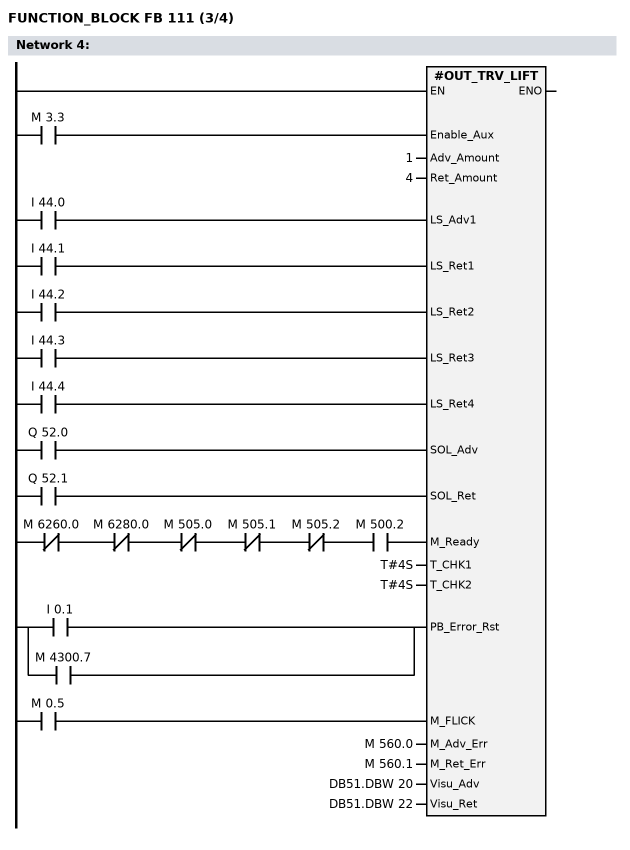

      A     M      3.3;
      =     L      0.0;
      BLD   103;
      A     I     44.0;
      =     L      0.1;
      BLD   103;
      A     I     44.1;
      =     L      0.2;
      BLD   103;
      A     I     44.2;
      =     L      0.4;
      BLD   103;
      A     I     44.3;
      =     L      0.6;
      BLD   103;
      A     I     44.4;
      =     L      1.0;
      BLD   103;
      A     Q     52.0;
      =     L      1.1;
      BLD   103;
      A     Q     52.1;
      =     L      1.2;
      BLD   103;
      AN    M   6260.0;
      AN    M   6280.0;
      AN    M    505.0;
      AN    M    505.1;
      AN    M    505.2;
      A     M    500.2;
      =     L      1.3;
      BLD   103;
      A(    ;
      O     I      0.1;
      O     M   4300.7;
      )     ;
      =     L      1.5;
      BLD   103;
      A     M      0.5;
      =     L      1.6;
      BLD   103;
      CALL #OUT_TRV_LIFT (
           Enable_Aux               := L      0.0,
           Adv_Amount               := 1,
           Ret_Amount               := 4,
           LS_Adv1                  := L      0.1,
           LS_Ret1                  := L      0.2,
           LS_Ret2                  := L      0.4,
           LS_Ret3                  := L      0.6,
           LS_Ret4                  := L      1.0,
           SOL_Adv                  := L      1.1,
           SOL_Ret                  := L      1.2,
           M_Ready                  := L      1.3,
           T_CHK1                   := T#4S,
           T_CHK2                   := T#4S,
           PB_Error_Rst             := L      1.5,
           M_FLICK                  := L      1.6,
           M_Adv_Err                := M    560.0,
           M_Ret_Err                := M    560.1,
           Visu_Adv                 := DB51.DBW   20,
           Visu_Ret                 := DB51.DBW   22);
      NOP   0;
NETWORK
TITLE =OUT TRV 급전이상 항시OFF
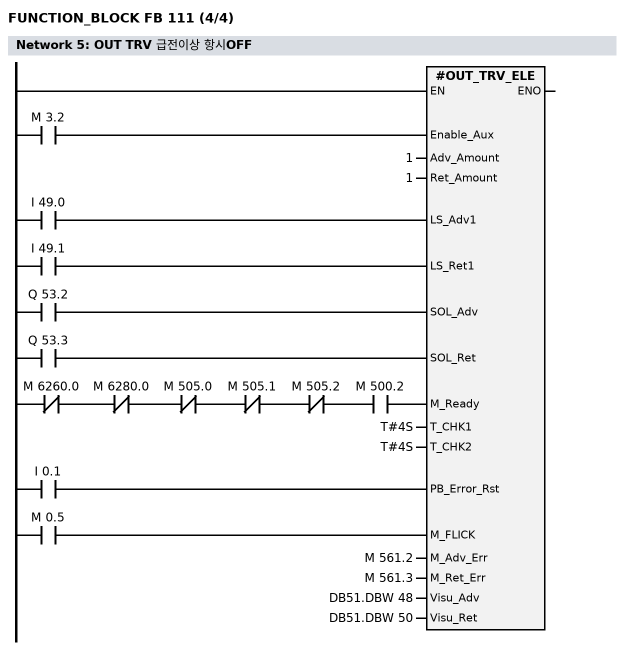

      A     M      3.2;
      =     L      0.0;
      BLD   103;
      A     I     49.0;
      =     L      0.1;
      BLD   103;
      A     I     49.1;
      =     L      0.2;
      BLD   103;
      A     Q     53.2;
      =     L      1.1;
      BLD   103;
      A     Q     53.3;
      =     L      1.2;
      BLD   103;
      AN    M   6260.0;
      AN    M   6280.0;
      AN    M    505.0;
      AN    M    505.1;
      AN    M    505.2;
      A     M    500.2;
      =     L      1.3;
      BLD   103;
      A     I      0.1;
      =     L      1.5;
      BLD   103;
      A     M      0.5;
      =     L      1.6;
      BLD   103;
      CALL #OUT_TRV_ELE (
           Enable_Aux               := L      0.0,
           Adv_Amount               := 1,
           Ret_Amount               := 1,
           LS_Adv1                  := L      0.1,
           LS_Ret1                  := L      0.2,
           SOL_Adv                  := L      1.1,
           SOL_Ret                  := L      1.2,
           M_Ready                  := L      1.3,
           T_CHK1                   := T#4S,
           T_CHK2                   := T#4S,
           PB_Error_Rst             := L      1.5,
           M_FLICK                  := L      1.6,
           M_Adv_Err                := M    561.2,
           M_Ret_Err                := M    561.3,
           Visu_Adv                 := DB51.DBW   48,
           Visu_Ret                 := DB51.DBW   50);
      NOP   0;
END_FUNCTION_BLOCK

DATA_BLOCK DB 111
TITLE =
VERSION : 0.0

 FB 111
BEGIN
   OUT_TRV_CUSHION_B.Enable_Aux := FALSE;
   OUT_TRV_CUSHION_B.Adv_Amount := 0;
   OUT_TRV_CUSHION_B.Ret_Amount := 0;
   OUT_TRV_CUSHION_B.LS_Adv1 := FALSE;
   OUT_TRV_CUSHION_B.LS_Ret1 := FALSE;
   OUT_TRV_CUSHION_B.LS_Adv2 := FALSE;
   OUT_TRV_CUSHION_B.LS_Ret2 := FALSE;
   OUT_TRV_CUSHION_B.LS_Adv3 := FALSE;
   OUT_TRV_CUSHION_B.LS_Ret3 := FALSE;
   OUT_TRV_CUSHION_B.LS_Adv4 := FALSE;
   OUT_TRV_CUSHION_B.LS_Ret4 := FALSE;
   OUT_TRV_CUSHION_B.SOL_Adv := FALSE;
   OUT_TRV_CUSHION_B.SOL_Ret := FALSE;
   OUT_TRV_CUSHION_B.M_Ready := FALSE;
   OUT_TRV_CUSHION_B.T_CHK1 := T#0MS;
   OUT_TRV_CUSHION_B.T_CHK2 := T#0MS;
   OUT_TRV_CUSHION_B.PB_Lamp_CHK := FALSE;
   OUT_TRV_CUSHION_B.PB_Error_Rst := FALSE;
   OUT_TRV_CUSHION_B.M_FLICK := FALSE;
   OUT_TRV_CUSHION_B.M_Adv_Err := FALSE;
   OUT_TRV_CUSHION_B.M_Ret_Err := FALSE;
   OUT_TRV_CUSHION_B.LP_Adv := FALSE;
   OUT_TRV_CUSHION_B.LP_Ret := FALSE;
   OUT_TRV_CUSHION_B.Visu_Adv := W#16#0;
   OUT_TRV_CUSHION_B.Visu_Ret := W#16#0;
   OUT_TRV_CUSHION_B.Error_T1.IN := FALSE;
   OUT_TRV_CUSHION_B.Error_T1.PT := T#0MS;
   OUT_TRV_CUSHION_B.Error_T1.Q := FALSE;
   OUT_TRV_CUSHION_B.Error_T1.ET := T#0MS;
   OUT_TRV_CUSHION_B.Error_T1.STATE := B#16#0;
   OUT_TRV_CUSHION_B.Error_T1.STIME := T#0MS;
   OUT_TRV_CUSHION_B.Error_T1.ATIME := T#0MS;
   OUT_TRV_CUSHION_B.Error_T2.IN := FALSE;
   OUT_TRV_CUSHION_B.Error_T2.PT := T#0MS;
   OUT_TRV_CUSHION_B.Error_T2.Q := FALSE;
   OUT_TRV_CUSHION_B.Error_T2.ET := T#0MS;
   OUT_TRV_CUSHION_B.Error_T2.STATE := B#16#0;
   OUT_TRV_CUSHION_B.Error_T2.STIME := T#0MS;
   OUT_TRV_CUSHION_B.Error_T2.ATIME := T#0MS;
   OUT_TRV_CUSHION_B.CHK_Aux1 := FALSE;
   OUT_TRV_CUSHION_B.CHK_Aux2 := FALSE;
   OUT_TRV_CUSHION_B.Error_T1_DN := FALSE;
   OUT_TRV_CUSHION_B.Error_T2_DN := FALSE;
   OUT_TRV_CUSHION_B.Adv_Memo := FALSE;
   OUT_TRV_CUSHION_B.Visu_Adv_Arr[0] := FALSE;
   OUT_TRV_CUSHION_B.Visu_Adv_Arr[1] := FALSE;
   OUT_TRV_CUSHION_B.Visu_Adv_Arr[2] := FALSE;
   OUT_TRV_CUSHION_B.Visu_Adv_Arr[3] := FALSE;
   OUT_TRV_CUSHION_B.Visu_Adv_Arr[4] := FALSE;
   OUT_TRV_CUSHION_B.Visu_Adv_Arr[5] := FALSE;
   OUT_TRV_CUSHION_B.Visu_Adv_Arr[6] := FALSE;
   OUT_TRV_CUSHION_B.Visu_Adv_Arr[7] := FALSE;
   OUT_TRV_CUSHION_B.Visu_Adv_Arr[8] := FALSE;
   OUT_TRV_CUSHION_B.Visu_Adv_Arr[9] := FALSE;
   OUT_TRV_CUSHION_B.Visu_Adv_Arr[10] := FALSE;
   OUT_TRV_CUSHION_B.Visu_Adv_Arr[11] := FALSE;
   OUT_TRV_CUSHION_B.Visu_Adv_Arr[12] := FALSE;
   OUT_TRV_CUSHION_B.Visu_Adv_Arr[13] := FALSE;
   OUT_TRV_CUSHION_B.Visu_Adv_Arr[14] := FALSE;
   OUT_TRV_CUSHION_B.Visu_Adv_Arr[15] := FALSE;
   OUT_TRV_CUSHION_B.Visu_Ret_Arr[0] := FALSE;
   OUT_TRV_CUSHION_B.Visu_Ret_Arr[1] := FALSE;
   OUT_TRV_CUSHION_B.Visu_Ret_Arr[2] := FALSE;
   OUT_TRV_CUSHION_B.Visu_Ret_Arr[3] := FALSE;
   OUT_TRV_CUSHION_B.Visu_Ret_Arr[4] := FALSE;
   OUT_TRV_CUSHION_B.Visu_Ret_Arr[5] := FALSE;
   OUT_TRV_CUSHION_B.Visu_Ret_Arr[6] := FALSE;
   OUT_TRV_CUSHION_B.Visu_Ret_Arr[7] := FALSE;
   OUT_TRV_CUSHION_B.Visu_Ret_Arr[8] := FALSE;
   OUT_TRV_CUSHION_B.Visu_Ret_Arr[9] := FALSE;
   OUT_TRV_CUSHION_B.Visu_Ret_Arr[10] := FALSE;
   OUT_TRV_CUSHION_B.Visu_Ret_Arr[11] := FALSE;
   OUT_TRV_CUSHION_B.Visu_Ret_Arr[12] := FALSE;
   OUT_TRV_CUSHION_B.Visu_Ret_Arr[13] := FALSE;
   OUT_TRV_CUSHION_B.Visu_Ret_Arr[14] := FALSE;
   OUT_TRV_CUSHION_B.Visu_Ret_Arr[15] := FALSE;
   OUT_TRV_CUSHION_B.BLK_Move_Ret := 0;
   OUT_TRV_CUSHION_B.Enable := FALSE;
   OUT_TRV_CUSHION_B.Adv_End := FALSE;
   OUT_TRV_CUSHION_B.Ret_End := FALSE;
   OUT_TRV_GUIDE.Enable_Aux := FALSE;
   OUT_TRV_GUIDE.Adv_Amount := 0;
   OUT_TRV_GUIDE.Ret_Amount := 0;
   OUT_TRV_GUIDE.LS_Adv1 := FALSE;
   OUT_TRV_GUIDE.LS_Ret1 := FALSE;
   OUT_TRV_GUIDE.LS_Adv2 := FALSE;
   OUT_TRV_GUIDE.LS_Ret2 := FALSE;
   OUT_TRV_GUIDE.LS_Adv3 := FALSE;
   OUT_TRV_GUIDE.LS_Ret3 := FALSE;
   OUT_TRV_GUIDE.LS_Adv4 := FALSE;
   OUT_TRV_GUIDE.LS_Ret4 := FALSE;
   OUT_TRV_GUIDE.SOL_Adv := FALSE;
   OUT_TRV_GUIDE.SOL_Ret := FALSE;
   OUT_TRV_GUIDE.M_Ready := FALSE;
   OUT_TRV_GUIDE.T_CHK1 := T#0MS;
   OUT_TRV_GUIDE.T_CHK2 := T#0MS;
   OUT_TRV_GUIDE.PB_Lamp_CHK := FALSE;
   OUT_TRV_GUIDE.PB_Error_Rst := FALSE;
   OUT_TRV_GUIDE.M_FLICK := FALSE;
   OUT_TRV_GUIDE.M_Adv_Err := FALSE;
   OUT_TRV_GUIDE.M_Ret_Err := FALSE;
   OUT_TRV_GUIDE.LP_Adv := FALSE;
   OUT_TRV_GUIDE.LP_Ret := FALSE;
   OUT_TRV_GUIDE.Visu_Adv := W#16#0;
   OUT_TRV_GUIDE.Visu_Ret := W#16#0;
   OUT_TRV_GUIDE.Error_T1.IN := FALSE;
   OUT_TRV_GUIDE.Error_T1.PT := T#0MS;
   OUT_TRV_GUIDE.Error_T1.Q := FALSE;
   OUT_TRV_GUIDE.Error_T1.ET := T#0MS;
   OUT_TRV_GUIDE.Error_T1.STATE := B#16#0;
   OUT_TRV_GUIDE.Error_T1.STIME := T#0MS;
   OUT_TRV_GUIDE.Error_T1.ATIME := T#0MS;
   OUT_TRV_GUIDE.Error_T2.IN := FALSE;
   OUT_TRV_GUIDE.Error_T2.PT := T#0MS;
   OUT_TRV_GUIDE.Error_T2.Q := FALSE;
   OUT_TRV_GUIDE.Error_T2.ET := T#0MS;
   OUT_TRV_GUIDE.Error_T2.STATE := B#16#0;
   OUT_TRV_GUIDE.Error_T2.STIME := T#0MS;
   OUT_TRV_GUIDE.Error_T2.ATIME := T#0MS;
   OUT_TRV_GUIDE.CHK_Aux1 := FALSE;
   OUT_TRV_GUIDE.CHK_Aux2 := FALSE;
   OUT_TRV_GUIDE.Error_T1_DN := FALSE;
   OUT_TRV_GUIDE.Error_T2_DN := FALSE;
   OUT_TRV_GUIDE.Adv_Memo := FALSE;
   OUT_TRV_GUIDE.Visu_Adv_Arr[0] := FALSE;
   OUT_TRV_GUIDE.Visu_Adv_Arr[1] := FALSE;
   OUT_TRV_GUIDE.Visu_Adv_Arr[2] := FALSE;
   OUT_TRV_GUIDE.Visu_Adv_Arr[3] := FALSE;
   OUT_TRV_GUIDE.Visu_Adv_Arr[4] := FALSE;
   OUT_TRV_GUIDE.Visu_Adv_Arr[5] := FALSE;
   OUT_TRV_GUIDE.Visu_Adv_Arr[6] := FALSE;
   OUT_TRV_GUIDE.Visu_Adv_Arr[7] := FALSE;
   OUT_TRV_GUIDE.Visu_Adv_Arr[8] := FALSE;
   OUT_TRV_GUIDE.Visu_Adv_Arr[9] := FALSE;
   OUT_TRV_GUIDE.Visu_Adv_Arr[10] := FALSE;
   OUT_TRV_GUIDE.Visu_Adv_Arr[11] := FALSE;
   OUT_TRV_GUIDE.Visu_Adv_Arr[12] := FALSE;
   OUT_TRV_GUIDE.Visu_Adv_Arr[13] := FALSE;
   OUT_TRV_GUIDE.Visu_Adv_Arr[14] := FALSE;
   OUT_TRV_GUIDE.Visu_Adv_Arr[15] := FALSE;
   OUT_TRV_GUIDE.Visu_Ret_Arr[0] := FALSE;
   OUT_TRV_GUIDE.Visu_Ret_Arr[1] := FALSE;
   OUT_TRV_GUIDE.Visu_Ret_Arr[2] := FALSE;
   OUT_TRV_GUIDE.Visu_Ret_Arr[3] := FALSE;
   OUT_TRV_GUIDE.Visu_Ret_Arr[4] := FALSE;
   OUT_TRV_GUIDE.Visu_Ret_Arr[5] := FALSE;
   OUT_TRV_GUIDE.Visu_Ret_Arr[6] := FALSE;
   OUT_TRV_GUIDE.Visu_Ret_Arr[7] := FALSE;
   OUT_TRV_GUIDE.Visu_Ret_Arr[8] := FALSE;
   OUT_TRV_GUIDE.Visu_Ret_Arr[9] := FALSE;
   OUT_TRV_GUIDE.Visu_Ret_Arr[10] := FALSE;
   OUT_TRV_GUIDE.Visu_Ret_Arr[11] := FALSE;
   OUT_TRV_GUIDE.Visu_Ret_Arr[12] := FALSE;
   OUT_TRV_GUIDE.Visu_Ret_Arr[13] := FALSE;
   OUT_TRV_GUIDE.Visu_Ret_Arr[14] := FALSE;
   OUT_TRV_GUIDE.Visu_Ret_Arr[15] := FALSE;
   OUT_TRV_GUIDE.BLK_Move_Ret := 0;
   OUT_TRV_GUIDE.Enable := FALSE;
   OUT_TRV_GUIDE.Adv_End := FALSE;
   OUT_TRV_GUIDE.Ret_End := FALSE;
   OUT_TRV_CLAMP.Enable_Aux := FALSE;
   OUT_TRV_CLAMP.Adv_Amount := 0;
   OUT_TRV_CLAMP.Ret_Amount := 0;
   OUT_TRV_CLAMP.LS_Adv1 := FALSE;
   OUT_TRV_CLAMP.LS_Ret1 := FALSE;
   OUT_TRV_CLAMP.LS_Adv2 := FALSE;
   OUT_TRV_CLAMP.LS_Ret2 := FALSE;
   OUT_TRV_CLAMP.LS_Adv3 := FALSE;
   OUT_TRV_CLAMP.LS_Ret3 := FALSE;
   OUT_TRV_CLAMP.LS_Adv4 := FALSE;
   OUT_TRV_CLAMP.LS_Ret4 := FALSE;
   OUT_TRV_CLAMP.SOL_Adv := FALSE;
   OUT_TRV_CLAMP.SOL_Ret := FALSE;
   OUT_TRV_CLAMP.M_Ready := FALSE;
   OUT_TRV_CLAMP.T_CHK1 := T#0MS;
   OUT_TRV_CLAMP.T_CHK2 := T#0MS;
   OUT_TRV_CLAMP.PB_Lamp_CHK := FALSE;
   OUT_TRV_CLAMP.PB_Error_Rst := FALSE;
   OUT_TRV_CLAMP.M_FLICK := FALSE;
   OUT_TRV_CLAMP.M_Adv_Err := FALSE;
   OUT_TRV_CLAMP.M_Ret_Err := FALSE;
   OUT_TRV_CLAMP.LP_Adv := FALSE;
   OUT_TRV_CLAMP.LP_Ret := FALSE;
   OUT_TRV_CLAMP.Visu_Adv := W#16#0;
   OUT_TRV_CLAMP.Visu_Ret := W#16#0;
   OUT_TRV_CLAMP.Error_T1.IN := FALSE;
   OUT_TRV_CLAMP.Error_T1.PT := T#0MS;
   OUT_TRV_CLAMP.Error_T1.Q := FALSE;
   OUT_TRV_CLAMP.Error_T1.ET := T#0MS;
   OUT_TRV_CLAMP.Error_T1.STATE := B#16#0;
   OUT_TRV_CLAMP.Error_T1.STIME := T#0MS;
   OUT_TRV_CLAMP.Error_T1.ATIME := T#0MS;
   OUT_TRV_CLAMP.Error_T2.IN := FALSE;
   OUT_TRV_CLAMP.Error_T2.PT := T#0MS;
   OUT_TRV_CLAMP.Error_T2.Q := FALSE;
   OUT_TRV_CLAMP.Error_T2.ET := T#0MS;
   OUT_TRV_CLAMP.Error_T2.STATE := B#16#0;
   OUT_TRV_CLAMP.Error_T2.STIME := T#0MS;
   OUT_TRV_CLAMP.Error_T2.ATIME := T#0MS;
   OUT_TRV_CLAMP.CHK_Aux1 := FALSE;
   OUT_TRV_CLAMP.CHK_Aux2 := FALSE;
   OUT_TRV_CLAMP.Error_T1_DN := FALSE;
   OUT_TRV_CLAMP.Error_T2_DN := FALSE;
   OUT_TRV_CLAMP.Adv_Memo := FALSE;
   OUT_TRV_CLAMP.Visu_Adv_Arr[0] := FALSE;
   OUT_TRV_CLAMP.Visu_Adv_Arr[1] := FALSE;
   OUT_TRV_CLAMP.Visu_Adv_Arr[2] := FALSE;
   OUT_TRV_CLAMP.Visu_Adv_Arr[3] := FALSE;
   OUT_TRV_CLAMP.Visu_Adv_Arr[4] := FALSE;
   OUT_TRV_CLAMP.Visu_Adv_Arr[5] := FALSE;
   OUT_TRV_CLAMP.Visu_Adv_Arr[6] := FALSE;
   OUT_TRV_CLAMP.Visu_Adv_Arr[7] := FALSE;
   OUT_TRV_CLAMP.Visu_Adv_Arr[8] := FALSE;
   OUT_TRV_CLAMP.Visu_Adv_Arr[9] := FALSE;
   OUT_TRV_CLAMP.Visu_Adv_Arr[10] := FALSE;
   OUT_TRV_CLAMP.Visu_Adv_Arr[11] := FALSE;
   OUT_TRV_CLAMP.Visu_Adv_Arr[12] := FALSE;
   OUT_TRV_CLAMP.Visu_Adv_Arr[13] := FALSE;
   OUT_TRV_CLAMP.Visu_Adv_Arr[14] := FALSE;
   OUT_TRV_CLAMP.Visu_Adv_Arr[15] := FALSE;
   OUT_TRV_CLAMP.Visu_Ret_Arr[0] := FALSE;
   OUT_TRV_CLAMP.Visu_Ret_Arr[1] := FALSE;
   OUT_TRV_CLAMP.Visu_Ret_Arr[2] := FALSE;
   OUT_TRV_CLAMP.Visu_Ret_Arr[3] := FALSE;
   OUT_TRV_CLAMP.Visu_Ret_Arr[4] := FALSE;
   OUT_TRV_CLAMP.Visu_Ret_Arr[5] := FALSE;
   OUT_TRV_CLAMP.Visu_Ret_Arr[6] := FALSE;
   OUT_TRV_CLAMP.Visu_Ret_Arr[7] := FALSE;
   OUT_TRV_CLAMP.Visu_Ret_Arr[8] := FALSE;
   OUT_TRV_CLAMP.Visu_Ret_Arr[9] := FALSE;
   OUT_TRV_CLAMP.Visu_Ret_Arr[10] := FALSE;
   OUT_TRV_CLAMP.Visu_Ret_Arr[11] := FALSE;
   OUT_TRV_CLAMP.Visu_Ret_Arr[12] := FALSE;
   OUT_TRV_CLAMP.Visu_Ret_Arr[13] := FALSE;
   OUT_TRV_CLAMP.Visu_Ret_Arr[14] := FALSE;
   OUT_TRV_CLAMP.Visu_Ret_Arr[15] := FALSE;
   OUT_TRV_CLAMP.BLK_Move_Ret := 0;
   OUT_TRV_CLAMP.Enable := FALSE;
   OUT_TRV_CLAMP.Adv_End := FALSE;
   OUT_TRV_CLAMP.Ret_End := FALSE;
   OUT_TRV_LIFT.Enable_Aux := FALSE;
   OUT_TRV_LIFT.Adv_Amount := 0;
   OUT_TRV_LIFT.Ret_Amount := 0;
   OUT_TRV_LIFT.LS_Adv1 := FALSE;
   OUT_TRV_LIFT.LS_Ret1 := FALSE;
   OUT_TRV_LIFT.LS_Adv2 := FALSE;
   OUT_TRV_LIFT.LS_Ret2 := FALSE;
   OUT_TRV_LIFT.LS_Adv3 := FALSE;
   OUT_TRV_LIFT.LS_Ret3 := FALSE;
   OUT_TRV_LIFT.LS_Adv4 := FALSE;
   OUT_TRV_LIFT.LS_Ret4 := FALSE;
   OUT_TRV_LIFT.SOL_Adv := FALSE;
   OUT_TRV_LIFT.SOL_Ret := FALSE;
   OUT_TRV_LIFT.M_Ready := FALSE;
   OUT_TRV_LIFT.T_CHK1 := T#0MS;
   OUT_TRV_LIFT.T_CHK2 := T#0MS;
   OUT_TRV_LIFT.PB_Lamp_CHK := FALSE;
   OUT_TRV_LIFT.PB_Error_Rst := FALSE;
   OUT_TRV_LIFT.M_FLICK := FALSE;
   OUT_TRV_LIFT.M_Adv_Err := FALSE;
   OUT_TRV_LIFT.M_Ret_Err := FALSE;
   OUT_TRV_LIFT.LP_Adv := FALSE;
   OUT_TRV_LIFT.LP_Ret := FALSE;
   OUT_TRV_LIFT.Visu_Adv := W#16#0;
   OUT_TRV_LIFT.Visu_Ret := W#16#0;
   OUT_TRV_LIFT.Error_T1.IN := FALSE;
   OUT_TRV_LIFT.Error_T1.PT := T#0MS;
   OUT_TRV_LIFT.Error_T1.Q := FALSE;
   OUT_TRV_LIFT.Error_T1.ET := T#0MS;
   OUT_TRV_LIFT.Error_T1.STATE := B#16#0;
   OUT_TRV_LIFT.Error_T1.STIME := T#0MS;
   OUT_TRV_LIFT.Error_T1.ATIME := T#0MS;
   OUT_TRV_LIFT.Error_T2.IN := FALSE;
   OUT_TRV_LIFT.Error_T2.PT := T#0MS;
   OUT_TRV_LIFT.Error_T2.Q := FALSE;
   OUT_TRV_LIFT.Error_T2.ET := T#0MS;
   OUT_TRV_LIFT.Error_T2.STATE := B#16#0;
   OUT_TRV_LIFT.Error_T2.STIME := T#0MS;
   OUT_TRV_LIFT.Error_T2.ATIME := T#0MS;
   OUT_TRV_LIFT.CHK_Aux1 := FALSE;
   OUT_TRV_LIFT.CHK_Aux2 := FALSE;
   OUT_TRV_LIFT.Error_T1_DN := FALSE;
   OUT_TRV_LIFT.Error_T2_DN := FALSE;
   OUT_TRV_LIFT.Adv_Memo := FALSE;
   OUT_TRV_LIFT.Visu_Adv_Arr[0] := FALSE;
   OUT_TRV_LIFT.Visu_Adv_Arr[1] := FALSE;
   OUT_TRV_LIFT.Visu_Adv_Arr[2] := FALSE;
   OUT_TRV_LIFT.Visu_Adv_Arr[3] := FALSE;
   OUT_TRV_LIFT.Visu_Adv_Arr[4] := FALSE;
   OUT_TRV_LIFT.Visu_Adv_Arr[5] := FALSE;
   OUT_TRV_LIFT.Visu_Adv_Arr[6] := FALSE;
   OUT_TRV_LIFT.Visu_Adv_Arr[7] := FALSE;
   OUT_TRV_LIFT.Visu_Adv_Arr[8] := FALSE;
   OUT_TRV_LIFT.Visu_Adv_Arr[9] := FALSE;
   OUT_TRV_LIFT.Visu_Adv_Arr[10] := FALSE;
   OUT_TRV_LIFT.Visu_Adv_Arr[11] := FALSE;
   OUT_TRV_LIFT.Visu_Adv_Arr[12] := FALSE;
   OUT_TRV_LIFT.Visu_Adv_Arr[13] := FALSE;
   OUT_TRV_LIFT.Visu_Adv_Arr[14] := FALSE;
   OUT_TRV_LIFT.Visu_Adv_Arr[15] := FALSE;
   OUT_TRV_LIFT.Visu_Ret_Arr[0] := FALSE;
   OUT_TRV_LIFT.Visu_Ret_Arr[1] := FALSE;
   OUT_TRV_LIFT.Visu_Ret_Arr[2] := FALSE;
   OUT_TRV_LIFT.Visu_Ret_Arr[3] := FALSE;
   OUT_TRV_LIFT.Visu_Ret_Arr[4] := FALSE;
   OUT_TRV_LIFT.Visu_Ret_Arr[5] := FALSE;
   OUT_TRV_LIFT.Visu_Ret_Arr[6] := FALSE;
   OUT_TRV_LIFT.Visu_Ret_Arr[7] := FALSE;
   OUT_TRV_LIFT.Visu_Ret_Arr[8] := FALSE;
   OUT_TRV_LIFT.Visu_Ret_Arr[9] := FALSE;
   OUT_TRV_LIFT.Visu_Ret_Arr[10] := FALSE;
   OUT_TRV_LIFT.Visu_Ret_Arr[11] := FALSE;
   OUT_TRV_LIFT.Visu_Ret_Arr[12] := FALSE;
   OUT_TRV_LIFT.Visu_Ret_Arr[13] := FALSE;
   OUT_TRV_LIFT.Visu_Ret_Arr[14] := FALSE;
   OUT_TRV_LIFT.Visu_Ret_Arr[15] := FALSE;
   OUT_TRV_LIFT.BLK_Move_Ret := 0;
   OUT_TRV_LIFT.Enable := FALSE;
   OUT_TRV_LIFT.Adv_End := FALSE;
   OUT_TRV_LIFT.Ret_End := FALSE;
   OUT_TRV_ELE.Enable_Aux := FALSE;
   OUT_TRV_ELE.Adv_Amount := 0;
   OUT_TRV_ELE.Ret_Amount := 0;
   OUT_TRV_ELE.LS_Adv1 := FALSE;
   OUT_TRV_ELE.LS_Ret1 := FALSE;
   OUT_TRV_ELE.LS_Adv2 := FALSE;
   OUT_TRV_ELE.LS_Ret2 := FALSE;
   OUT_TRV_ELE.LS_Adv3 := FALSE;
   OUT_TRV_ELE.LS_Ret3 := FALSE;
   OUT_TRV_ELE.LS_Adv4 := FALSE;
   OUT_TRV_ELE.LS_Ret4 := FALSE;
   OUT_TRV_ELE.SOL_Adv := FALSE;
   OUT_TRV_ELE.SOL_Ret := FALSE;
   OUT_TRV_ELE.M_Ready := FALSE;
   OUT_TRV_ELE.T_CHK1 := T#0MS;
   OUT_TRV_ELE.T_CHK2 := T#0MS;
   OUT_TRV_ELE.PB_Lamp_CHK := FALSE;
   OUT_TRV_ELE.PB_Error_Rst := FALSE;
   OUT_TRV_ELE.M_FLICK := FALSE;
   OUT_TRV_ELE.M_Adv_Err := FALSE;
   OUT_TRV_ELE.M_Ret_Err := FALSE;
   OUT_TRV_ELE.LP_Adv := FALSE;
   OUT_TRV_ELE.LP_Ret := FALSE;
   OUT_TRV_ELE.Visu_Adv := W#16#0;
   OUT_TRV_ELE.Visu_Ret := W#16#0;
   OUT_TRV_ELE.Error_T1.IN := FALSE;
   OUT_TRV_ELE.Error_T1.PT := T#0MS;
   OUT_TRV_ELE.Error_T1.Q := FALSE;
   OUT_TRV_ELE.Error_T1.ET := T#0MS;
   OUT_TRV_ELE.Error_T1.STATE := B#16#0;
   OUT_TRV_ELE.Error_T1.STIME := T#0MS;
   OUT_TRV_ELE.Error_T1.ATIME := T#0MS;
   OUT_TRV_ELE.Error_T2.IN := FALSE;
   OUT_TRV_ELE.Error_T2.PT := T#0MS;
   OUT_TRV_ELE.Error_T2.Q := FALSE;
   OUT_TRV_ELE.Error_T2.ET := T#0MS;
   OUT_TRV_ELE.Error_T2.STATE := B#16#0;
   OUT_TRV_ELE.Error_T2.STIME := T#0MS;
   OUT_TRV_ELE.Error_T2.ATIME := T#0MS;
   OUT_TRV_ELE.CHK_Aux1 := FALSE;
   OUT_TRV_ELE.CHK_Aux2 := FALSE;
   OUT_TRV_ELE.Error_T1_DN := FALSE;
   OUT_TRV_ELE.Error_T2_DN := FALSE;
   OUT_TRV_ELE.Adv_Memo := FALSE;
   OUT_TRV_ELE.Visu_Adv_Arr[0] := FALSE;
   OUT_TRV_ELE.Visu_Adv_Arr[1] := FALSE;
   OUT_TRV_ELE.Visu_Adv_Arr[2] := FALSE;
   OUT_TRV_ELE.Visu_Adv_Arr[3] := FALSE;
   OUT_TRV_ELE.Visu_Adv_Arr[4] := FALSE;
   OUT_TRV_ELE.Visu_Adv_Arr[5] := FALSE;
   OUT_TRV_ELE.Visu_Adv_Arr[6] := FALSE;
   OUT_TRV_ELE.Visu_Adv_Arr[7] := FALSE;
   OUT_TRV_ELE.Visu_Adv_Arr[8] := FALSE;
   OUT_TRV_ELE.Visu_Adv_Arr[9] := FALSE;
   OUT_TRV_ELE.Visu_Adv_Arr[10] := FALSE;
   OUT_TRV_ELE.Visu_Adv_Arr[11] := FALSE;
   OUT_TRV_ELE.Visu_Adv_Arr[12] := FALSE;
   OUT_TRV_ELE.Visu_Adv_Arr[13] := FALSE;
   OUT_TRV_ELE.Visu_Adv_Arr[14] := FALSE;
   OUT_TRV_ELE.Visu_Adv_Arr[15] := FALSE;
   OUT_TRV_ELE.Visu_Ret_Arr[0] := FALSE;
   OUT_TRV_ELE.Visu_Ret_Arr[1] := FALSE;
   OUT_TRV_ELE.Visu_Ret_Arr[2] := FALSE;
   OUT_TRV_ELE.Visu_Ret_Arr[3] := FALSE;
   OUT_TRV_ELE.Visu_Ret_Arr[4] := FALSE;
   OUT_TRV_ELE.Visu_Ret_Arr[5] := FALSE;
   OUT_TRV_ELE.Visu_Ret_Arr[6] := FALSE;
   OUT_TRV_ELE.Visu_Ret_Arr[7] := FALSE;
   OUT_TRV_ELE.Visu_Ret_Arr[8] := FALSE;
   OUT_TRV_ELE.Visu_Ret_Arr[9] := FALSE;
   OUT_TRV_ELE.Visu_Ret_Arr[10] := FALSE;
   OUT_TRV_ELE.Visu_Ret_Arr[11] := FALSE;
   OUT_TRV_ELE.Visu_Ret_Arr[12] := FALSE;
   OUT_TRV_ELE.Visu_Ret_Arr[13] := FALSE;
   OUT_TRV_ELE.Visu_Ret_Arr[14] := FALSE;
   OUT_TRV_ELE.Visu_Ret_Arr[15] := FALSE;
   OUT_TRV_ELE.BLK_Move_Ret := 0;
   OUT_TRV_ELE.Enable := FALSE;
   OUT_TRV_ELE.Adv_End := FALSE;
   OUT_TRV_ELE.Ret_End := FALSE;
END_DATA_BLOCK

FUNCTION FC 111 : VOID
TITLE =
VERSION : 0.1

BEGIN
NETWORK
TITLE =
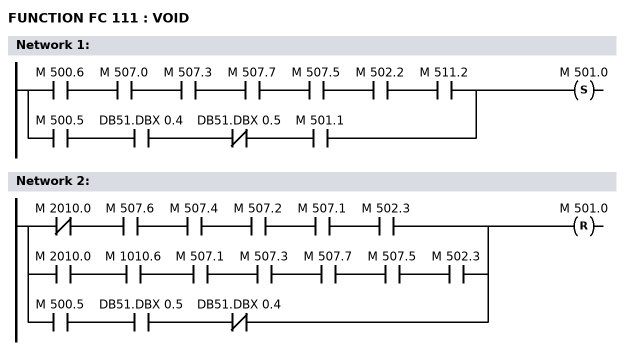

      A     M    500.6;
      A     M    507.0;
      A     M    507.3;
      A     M    507.7;
      A     M    507.5;
      A     M    502.2;
      A     M    511.2;
      O     ;
      A     M    500.5;
      A     DB51.DBX    0.4;
      AN    DB51.DBX    0.5;
      A     M    501.1;
      S     M    501.0;
NETWORK
TITLE =

      AN    M   2010.0;
      A     M    507.6;
      A     M    507.4;
      A     M    507.2;
      A     M    507.1;
      A     M    502.3;
      O     ;
      A     M   2010.0;
      A     M   1010.6;
      A     M    507.1;
      A     M    507.3;
      A     M    507.7;
      A     M    507.5;
      A     M    502.3;
      O     ;
      A     M    500.5;
      A     DB51.DBX    0.5;
      AN    DB51.DBX    0.4;
      R     M    501.0;
END_FUNCTION

FUNCTION_BLOCK FB 112
TITLE =
VERSION : 0.1

BEGIN
NETWORK
TITLE =
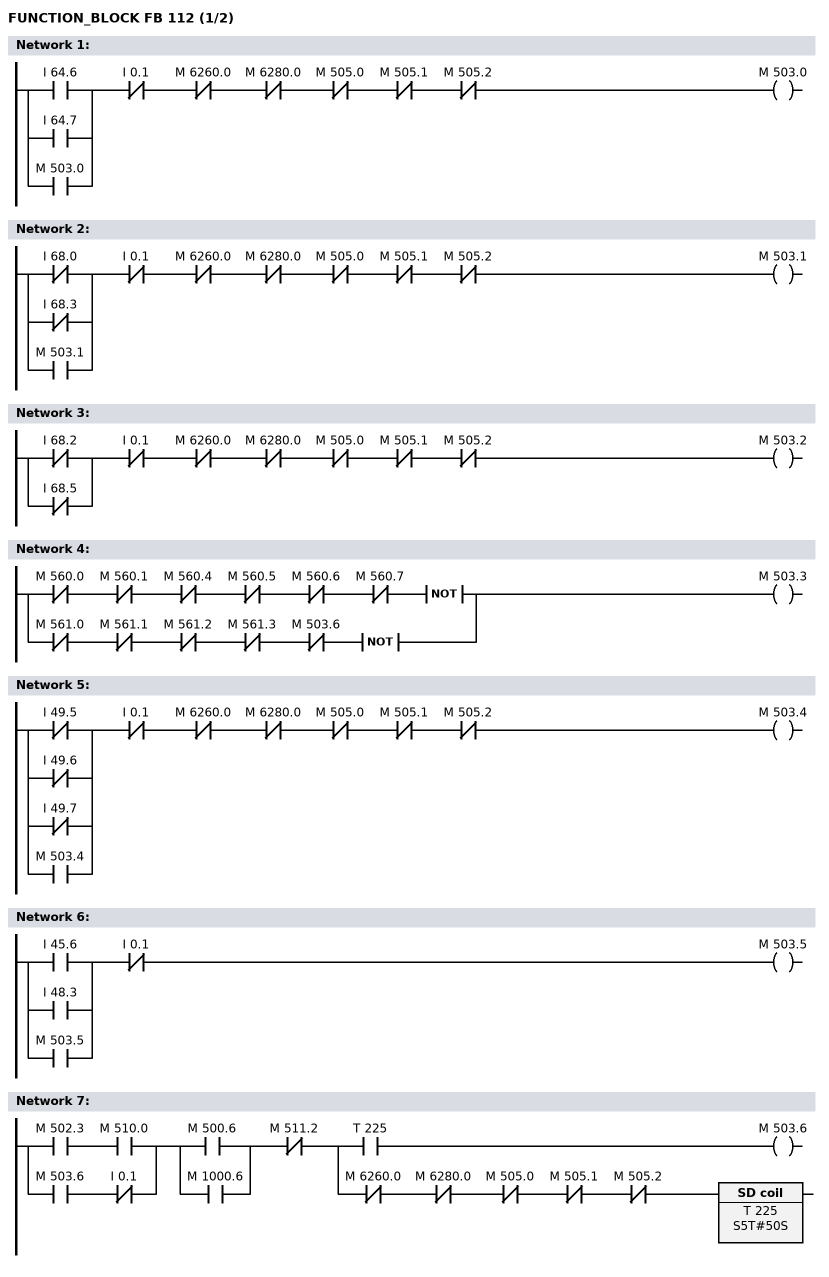

      A(    ;
      O     I     64.6;
      O     I     64.7;
      O     M    503.0;
      )     ;
      AN    I      0.1;
      AN    M   6260.0;
      AN    M   6280.0;
      AN    M    505.0;
      AN    M    505.1;
      AN    M    505.2;
      =     M    503.0;
NETWORK
TITLE =

      A(    ;
      ON    I     68.0;
      ON    I     68.3;
      O     M    503.1;
      )     ;
      AN    I      0.1;
      AN    M   6260.0;
      AN    M   6280.0;
      AN    M    505.0;
      AN    M    505.1;
      AN    M    505.2;
      =     M    503.1;
NETWORK
TITLE =

      A(    ;
      ON    I     68.2;
      ON    I     68.5;
      )     ;
      AN    I      0.1;
      AN    M   6260.0;
      AN    M   6280.0;
      AN    M    505.0;
      AN    M    505.1;
      AN    M    505.2;
      =     M    503.2;
NETWORK
TITLE =

      AN    M    560.0;
      AN    M    560.1;
      AN    M    560.4;
      AN    M    560.5;
      AN    M    560.6;
      AN    M    560.7;
      NOT   ;
      O(    ;
      AN    M    561.0;
      AN    M    561.1;
      AN    M    561.2;
      AN    M    561.3;
      AN    M    503.6;
      NOT   ;
      )     ;
      =     M    503.3;
NETWORK
TITLE =

      A(    ;
      ON    I     49.5;
      ON    I     49.6;
      ON    I     49.7;
      O     M    503.4;
      )     ;
      AN    I      0.1;
      AN    M   6260.0;
      AN    M   6280.0;
      AN    M    505.0;
      AN    M    505.1;
      AN    M    505.2;
      =     M    503.4;
NETWORK
TITLE =

      A(    ;
      O     I     45.6;
      O     I     48.3;
      O     M    503.5;
      )     ;
      AN    I      0.1;
      =     M    503.5;
NETWORK
TITLE =

      A(    ;
      A     M    502.3;
      A     M    510.0;
      O     ;
      A     M    503.6;
      AN    I      0.1;
      )     ;
      A(    ;
      O     M    500.6;
      O     M   1000.6;
      )     ;
      AN    M    511.2;
      =     L      0.0;
      A     L      0.0;
      A     T    225;
      =     M    503.6;
      A     L      0.0;
      AN    M   6260.0;
      AN    M   6280.0;
      AN    M    505.0;
      AN    M    505.1;
      AN    M    505.2;
      L     S5T#50S;
      SD    T    225;
NETWORK
TITLE =
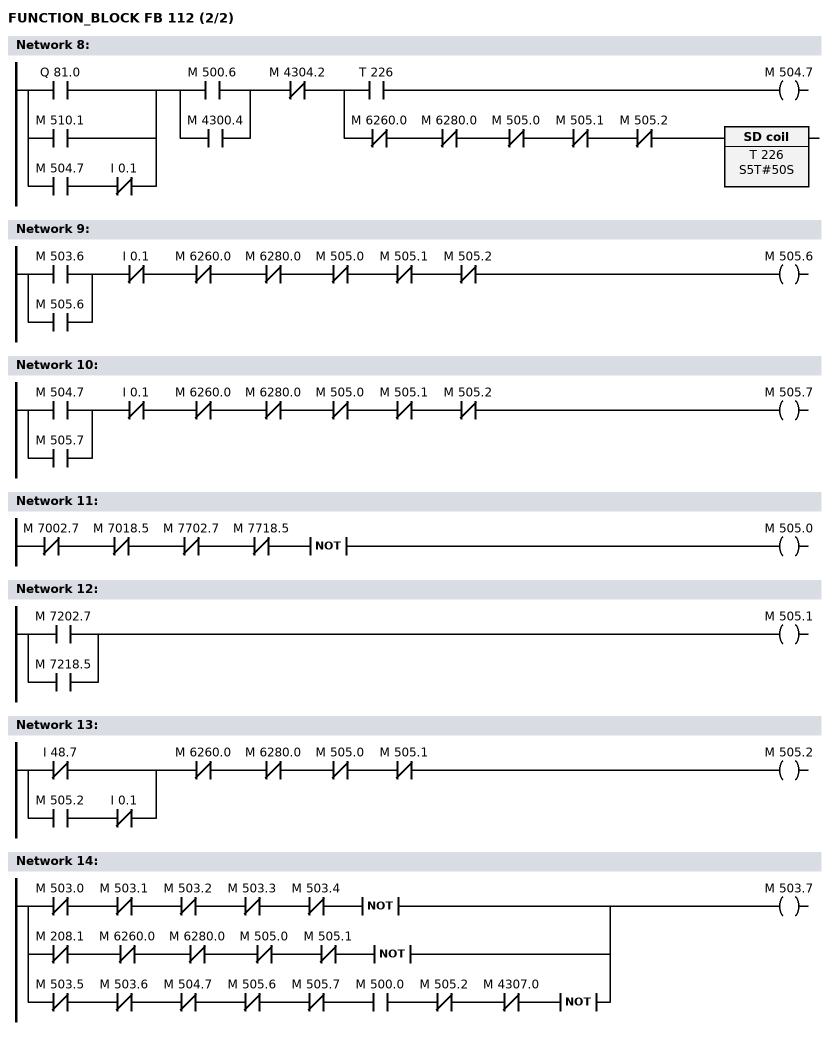

      A(    ;
      O     Q     81.0;
      O     M    510.1;
      O     ;
      A     M    504.7;
      AN    I      0.1;
      )     ;
      A(    ;
      O     M    500.6;
      O     M   4300.4;
      )     ;
      AN    M   4304.2;
      =     L      0.0;
      A     L      0.0;
      A     T    226;
      =     M    504.7;
      A     L      0.0;
      AN    M   6260.0;
      AN    M   6280.0;
      AN    M    505.0;
      AN    M    505.1;
      AN    M    505.2;
      L     S5T#50S;
      SD    T    226;
NETWORK
TITLE =

      A(    ;
      O     M    503.6;
      O     M    505.6;
      )     ;
      AN    I      0.1;
      AN    M   6260.0;
      AN    M   6280.0;
      AN    M    505.0;
      AN    M    505.1;
      AN    M    505.2;
      =     M    505.6;
NETWORK
TITLE =

      A(    ;
      O     M    504.7;
      O     M    505.7;
      )     ;
      AN    I      0.1;
      AN    M   6260.0;
      AN    M   6280.0;
      AN    M    505.0;
      AN    M    505.1;
      AN    M    505.2;
      =     M    505.7;
NETWORK
TITLE =

      AN    M   7002.7;
      AN    M   7018.5;
      AN    M   7702.7;
      AN    M   7718.5;
      NOT   ;
      =     M    505.0;
NETWORK
TITLE =

      O     M   7202.7;
      O     M   7218.5;
      =     M    505.1;
NETWORK
TITLE =

      A(    ;
      ON    I     48.7;
      O     ;
      A     M    505.2;
      AN    I      0.1;
      )     ;
      AN    M   6260.0;
      AN    M   6280.0;
      AN    M    505.0;
      AN    M    505.1;
      =     M    505.2;
NETWORK
TITLE =

      AN    M    503.0;
      AN    M    503.1;
      AN    M    503.2;
      AN    M    503.3;
      AN    M    503.4;
      NOT   ;
      O(    ;
      AN    M    208.1;
      AN    M   6260.0;
      AN    M   6280.0;
      AN    M    505.0;
      AN    M    505.1;
      NOT   ;
      )     ;
      O(    ;
      AN    M    503.5;
      AN    M    503.6;
      AN    M    504.7;
      AN    M    505.6;
      AN    M    505.7;
      A     M    500.0;
      AN    M    505.2;
      AN    M   4307.0;
      NOT   ;
      )     ;
      =     M    503.7;
END_FUNCTION_BLOCK

DATA_BLOCK DB 112
TITLE =
VERSION : 0.0

 FB 112
BEGIN
END_DATA_BLOCK

FUNCTION FC 112 : VOID
TITLE =
VERSION : 0.1

BEGIN
NETWORK
TITLE =
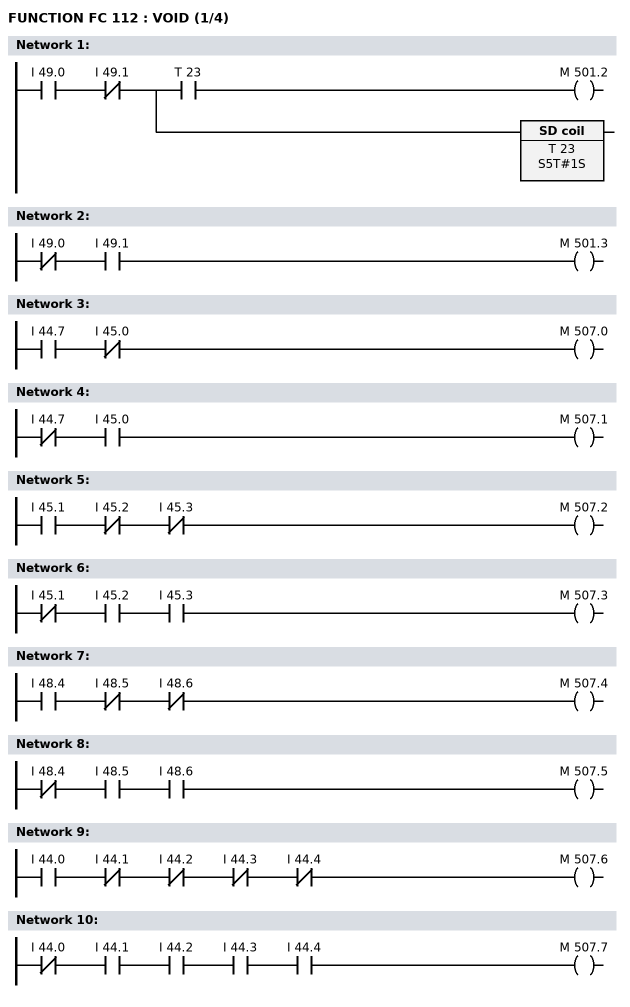

      A     I     49.0;
      AN    I     49.1;
      =     L      0.0;
      A     L      0.0;
      A     T     23;
      =     M    501.2;
      A     L      0.0;
      BLD   102;
      L     S5T#1S;
      SD    T     23;
NETWORK
TITLE =

      AN    I     49.0;
      A     I     49.1;
      =     M    501.3;
NETWORK
TITLE =

      A     I     44.7;
      AN    I     45.0;
      =     M    507.0;
NETWORK
TITLE =

      AN    I     44.7;
      A     I     45.0;
      =     M    507.1;
NETWORK
TITLE =

      A     I     45.1;
      AN    I     45.2;
      AN    I     45.3;
      =     M    507.2;
NETWORK
TITLE =

      AN    I     45.1;
      A     I     45.2;
      A     I     45.3;
      =     M    507.3;
NETWORK
TITLE =

      A     I     48.4;
      AN    I     48.5;
      AN    I     48.6;
      =     M    507.4;
NETWORK
TITLE =

      AN    I     48.4;
      A     I     48.5;
      A     I     48.6;
      =     M    507.5;
NETWORK
TITLE =

      A     I     44.0;
      AN    I     44.1;
      AN    I     44.2;
      AN    I     44.3;
      AN    I     44.4;
      =     M    507.6;
NETWORK
TITLE =

      AN    I     44.0;
      A     I     44.1;
      A     I     44.2;
      A     I     44.3;
      A     I     44.4;
      =     M    507.7;
NETWORK
TITLE =
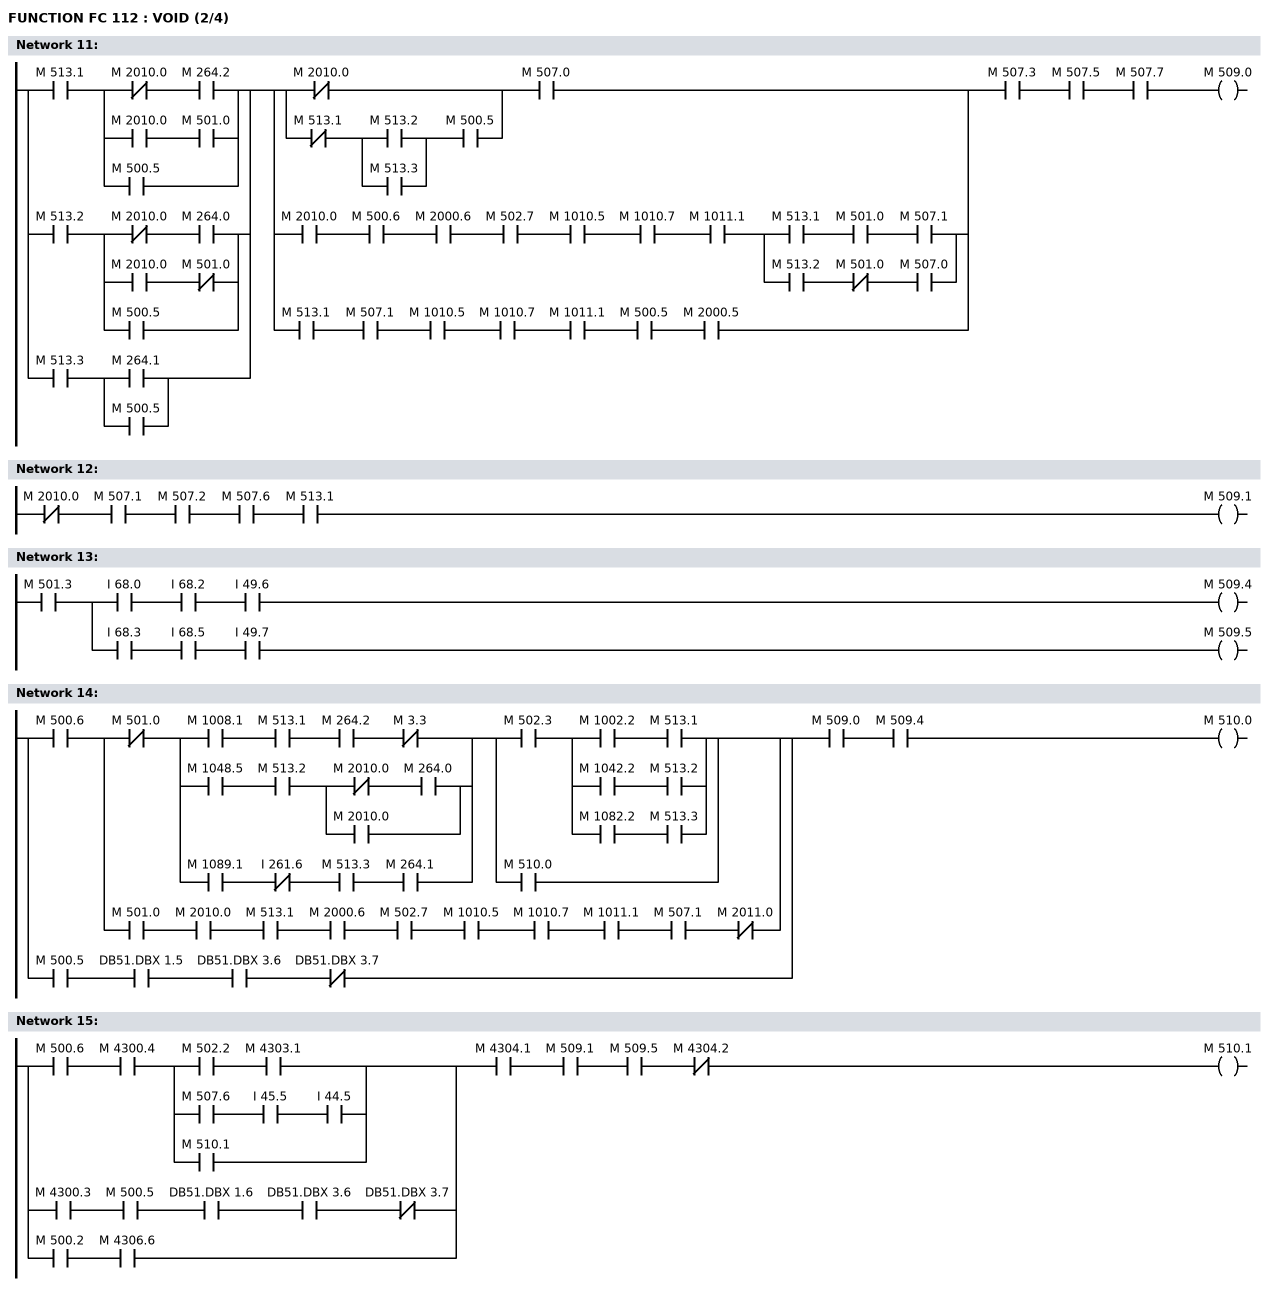

      A(    ;
      A     M    513.1;
      A(    ;
      AN    M   2010.0;
      A     M    264.2;
      O     ;
      A     M   2010.0;
      A     M    501.0;
      O     M    500.5;
      )     ;
      O     ;
      A     M    513.2;
      A(    ;
      AN    M   2010.0;
      A     M    264.0;
      O     ;
      A     M   2010.0;
      AN    M    501.0;
      O     M    500.5;
      )     ;
      O     ;
      A     M    513.3;
      A(    ;
      O     M    264.1;
      O     M    500.5;
      )     ;
      )     ;
      A(    ;
      A(    ;
      ON    M   2010.0;
      O     ;
      AN    M    513.1;
      A(    ;
      O     M    513.2;
      O     M    513.3;
      )     ;
      A     M    500.5;
      )     ;
      A     M    507.0;
      O     ;
      A     M   2010.0;
      A     M    500.6;
      A     M   2000.6;
      A     M    502.7;
      A     M   1010.5;
      A     M   1010.7;
      A     M   1011.1;
      A(    ;
      A     M    513.1;
      A     M    501.0;
      A     M    507.1;
      O     ;
      A     M    513.2;
      AN    M    501.0;
      A     M    507.0;
      )     ;
      O     ;
      A     M    513.1;
      A     M    507.1;
      A     M   1010.5;
      A     M   1010.7;
      A     M   1011.1;
      A     M    500.5;
      A     M   2000.5;
      )     ;
      A     M    507.3;
      A     M    507.5;
      A     M    507.7;
      =     M    509.0;
NETWORK
TITLE =

      AN    M   2010.0;
      A     M    507.1;
      A     M    507.2;
      A     M    507.6;
      A     M    513.1;
      =     M    509.1;
NETWORK
TITLE =

      A     M    501.3;
      =     L      0.0;
      A     L      0.0;
      A     I     68.0;
      A     I     68.2;
      A     I     49.6;
      =     M    509.4;
      A     L      0.0;
      A     I     68.3;
      A     I     68.5;
      A     I     49.7;
      =     M    509.5;
NETWORK
TITLE =

      A(    ;
      A     M    500.6;
      A(    ;
      AN    M    501.0;
      A(    ;
      A     M   1008.1;
      A     M    513.1;
      A     M    264.2;
      AN    M      3.3;
      O     ;
      A     M   1048.5;
      A     M    513.2;
      A(    ;
      AN    M   2010.0;
      A     M    264.0;
      O     M   2010.0;
      )     ;
      O     ;
      A     M   1089.1;
      AN    I    261.6;
      A     M    513.3;
      A     M    264.1;
      )     ;
      A(    ;
      A     M    502.3;
      A(    ;
      A     M   1002.2;
      A     M    513.1;
      O     ;
      A     M   1042.2;
      A     M    513.2;
      O     ;
      A     M   1082.2;
      A     M    513.3;
      )     ;
      O     M    510.0;
      )     ;
      O     ;
      A     M    501.0;
      A     M   2010.0;
      A     M    513.1;
      A     M   2000.6;
      A     M    502.7;
      A     M   1010.5;
      A     M   1010.7;
      A     M   1011.1;
      A     M    507.1;
      AN    M   2011.0;
      )     ;
      O     ;
      A     M    500.5;
      A     DB51.DBX    1.5;
      A     DB51.DBX    3.6;
      AN    DB51.DBX    3.7;
      )     ;
      A     M    509.0;
      A     M    509.4;
      =     M    510.0;
NETWORK
TITLE =

      A(    ;
      A     M    500.6;
      A     M   4300.4;
      A(    ;
      A     M    502.2;
      A     M   4303.1;
      O     ;
      A     M    507.6;
      A     I     45.5;
      A     I     44.5;
      O     M    510.1;
      )     ;
      O     ;
      A     M   4300.3;
      A     M    500.5;
      A     DB51.DBX    1.6;
      A     DB51.DBX    3.6;
      AN    DB51.DBX    3.7;
      O     ;
      A     M    500.2;
      A     M   4306.6;
      )     ;
      A     M   4304.1;
      A     M    509.1;
      A     M    509.5;
      AN    M   4304.2;
      =     M    510.1;
NETWORK
TITLE =
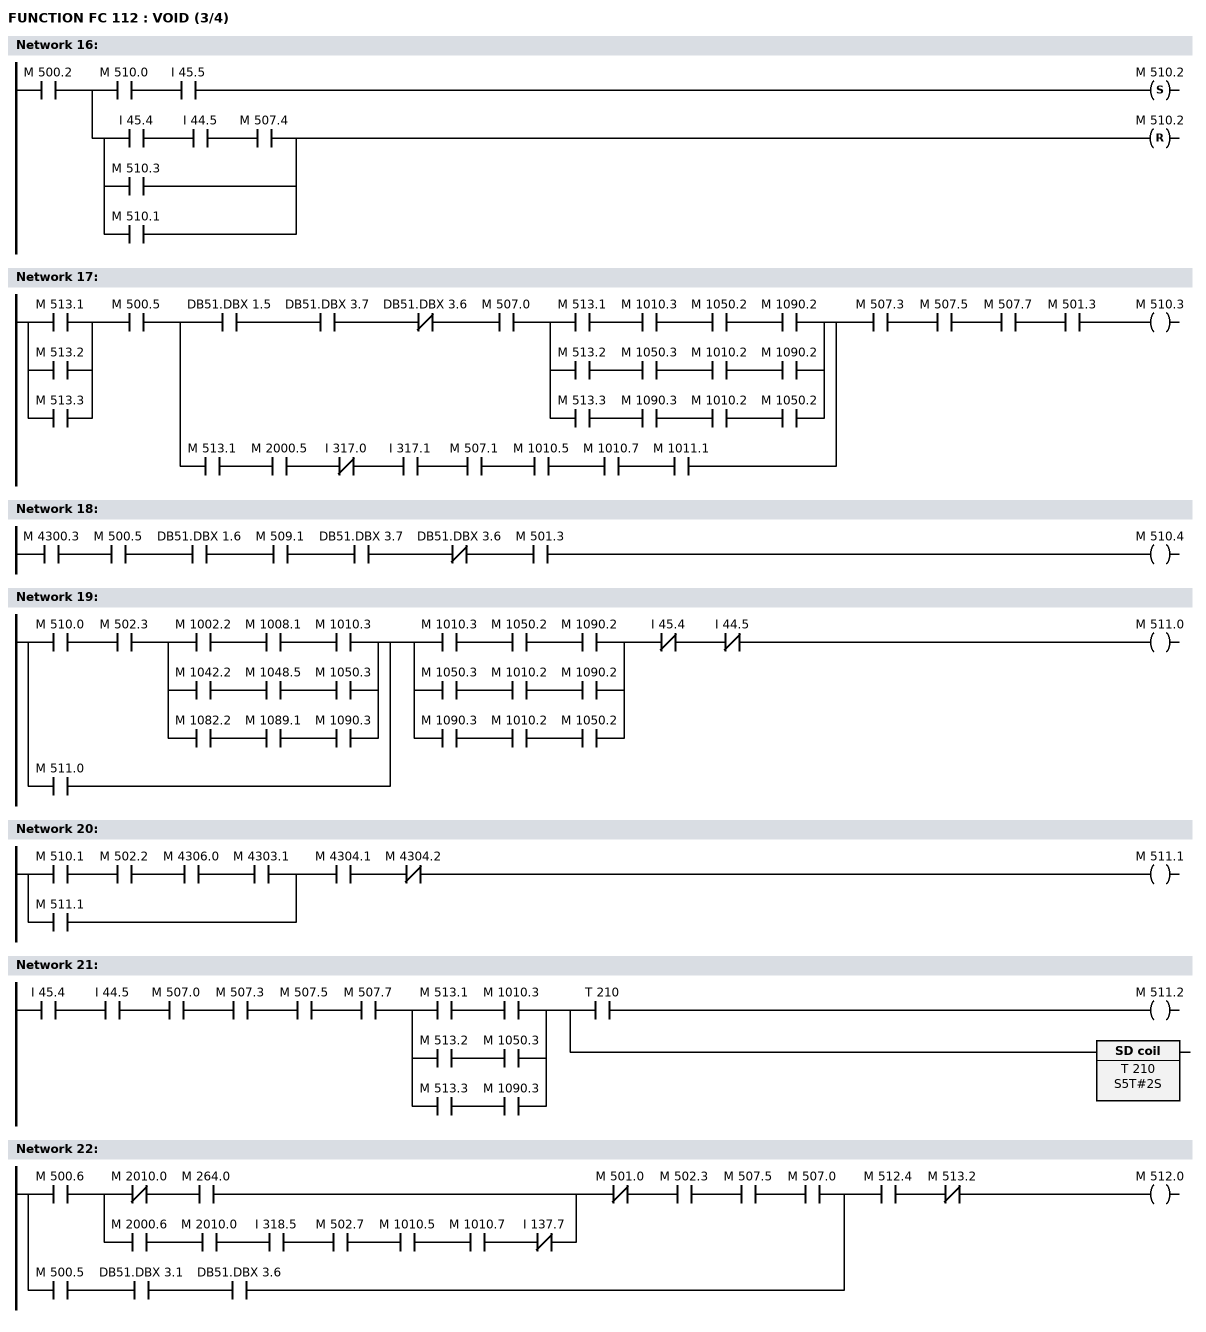

      A     M    500.2;
      =     L      0.0;
      A     L      0.0;
      A     M    510.0;
      A     I     45.5;
      S     M    510.2;
      A     L      0.0;
      A(    ;
      A     I     45.4;
      A     I     44.5;
      A     M    507.4;
      O     M    510.3;
      O     M    510.1;
      )     ;
      R     M    510.2;
NETWORK
TITLE =

      A(    ;
      O     M    513.1;
      O     M    513.2;
      O     M    513.3;
      )     ;
      A     M    500.5;
      A(    ;
      A     DB51.DBX    1.5;
      A     DB51.DBX    3.7;
      AN    DB51.DBX    3.6;
      A     M    507.0;
      A(    ;
      A     M    513.1;
      A     M   1010.3;
      A     M   1050.2;
      A     M   1090.2;
      O     ;
      A     M    513.2;
      A     M   1050.3;
      A     M   1010.2;
      A     M   1090.2;
      O     ;
      A     M    513.3;
      A     M   1090.3;
      A     M   1010.2;
      A     M   1050.2;
      )     ;
      O     ;
      A     M    513.1;
      A     M   2000.5;
      AN    I    317.0;
      A     I    317.1;
      A     M    507.1;
      A     M   1010.5;
      A     M   1010.7;
      A     M   1011.1;
      )     ;
      A     M    507.3;
      A     M    507.5;
      A     M    507.7;
      A     M    501.3;
      =     M    510.3;
NETWORK
TITLE =

      A     M   4300.3;
      A     M    500.5;
      A     DB51.DBX    1.6;
      A     M    509.1;
      A     DB51.DBX    3.7;
      AN    DB51.DBX    3.6;
      A     M    501.3;
      =     M    510.4;
NETWORK
TITLE =

      A(    ;
      A     M    510.0;
      A     M    502.3;
      A(    ;
      A     M   1002.2;
      A     M   1008.1;
      A     M   1010.3;
      O     ;
      A     M   1042.2;
      A     M   1048.5;
      A     M   1050.3;
      O     ;
      A     M   1082.2;
      A     M   1089.1;
      A     M   1090.3;
      )     ;
      O     M    511.0;
      )     ;
      A(    ;
      A     M   1010.3;
      A     M   1050.2;
      A     M   1090.2;
      O     ;
      A     M   1050.3;
      A     M   1010.2;
      A     M   1090.2;
      O     ;
      A     M   1090.3;
      A     M   1010.2;
      A     M   1050.2;
      )     ;
      AN    I     45.4;
      AN    I     44.5;
      =     M    511.0;
NETWORK
TITLE =

      A(    ;
      A     M    510.1;
      A     M    502.2;
      A     M   4306.0;
      A     M   4303.1;
      O     M    511.1;
      )     ;
      A     M   4304.1;
      AN    M   4304.2;
      =     M    511.1;
NETWORK
TITLE =

      A     I     45.4;
      A     I     44.5;
      A     M    507.0;
      A     M    507.3;
      A     M    507.5;
      A     M    507.7;
      A(    ;
      A     M    513.1;
      A     M   1010.3;
      O     ;
      A     M    513.2;
      A     M   1050.3;
      O     ;
      A     M    513.3;
      A     M   1090.3;
      )     ;
      =     L      0.0;
      A     L      0.0;
      A     T    210;
      =     M    511.2;
      A     L      0.0;
      BLD   102;
      L     S5T#2S;
      SD    T    210;
NETWORK
TITLE =

      A(    ;
      A     M    500.6;
      A(    ;
      AN    M   2010.0;
      A     M    264.0;
      O     ;
      A     M   2000.6;
      A     M   2010.0;
      A     I    318.5;
      A     M    502.7;
      A     M   1010.5;
      A     M   1010.7;
      AN    I    137.7;
      )     ;
      AN    M    501.0;
      A     M    502.3;
      A     M    507.5;
      A     M    507.0;
      O     ;
      A     M    500.5;
      A     DB51.DBX    3.1;
      A     DB51.DBX    3.6;
      )     ;
      A     M    512.4;
      AN    M    513.2;
      =     M    512.0;
NETWORK
TITLE =
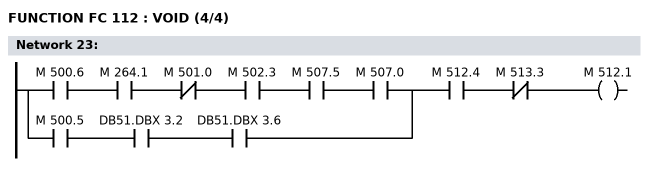

      A(    ;
      A     M    500.6;
      A     M    264.1;
      AN    M    501.0;
      A     M    502.3;
      A     M    507.5;
      A     M    507.0;
      O     ;
      A     M    500.5;
      A     DB51.DBX    3.2;
      A     DB51.DBX    3.6;
      )     ;
      A     M    512.4;
      AN    M    513.3;
      =     M    512.1;
NETWORK
TITLE =

      A     M    500.5;
      A     DB51.DBX    3.3;
      A     DB51.DBX    3.6;
      A     M    512.4;
      AN    M    513.4;
      A     OV;
      =     M    512.2;
NETWORK
TITLE =
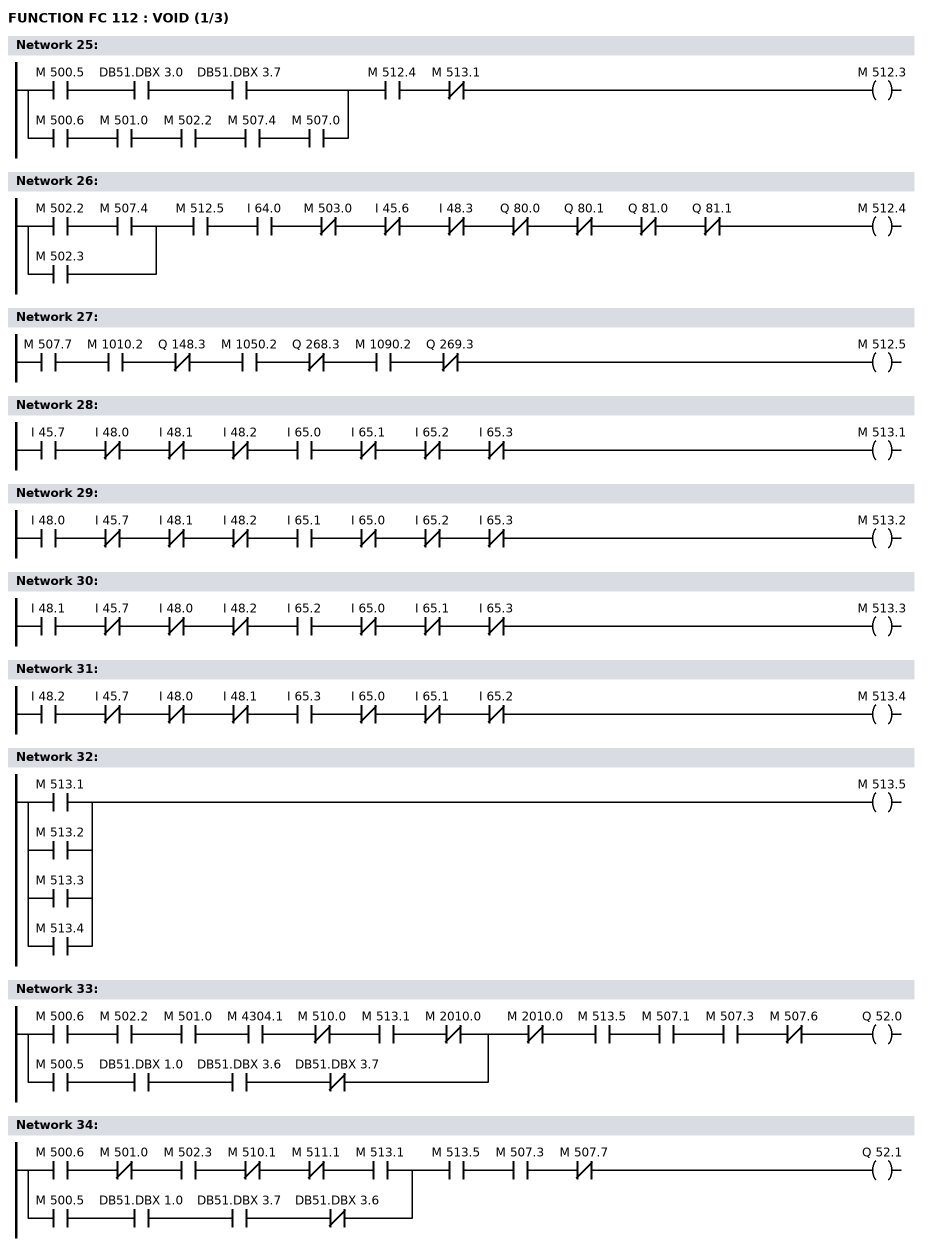

      A(    ;
      A     M    500.5;
      A     DB51.DBX    3.0;
      A     DB51.DBX    3.7;
      O     ;
      A     M    500.6;
      A     M    501.0;
      A     M    502.2;
      A     M    507.4;
      A     M    507.0;
      )     ;
      A     M    512.4;
      AN    M    513.1;
      =     M    512.3;
NETWORK
TITLE =

      A(    ;
      A     M    502.2;
      A     M    507.4;
      O     M    502.3;
      )     ;
      A     M    512.5;
      A     I     64.0;
      AN    M    503.0;
      AN    I     45.6;
      AN    I     48.3;
      AN    Q     80.0;
      AN    Q     80.1;
      AN    Q     81.0;
      AN    Q     81.1;
      =     M    512.4;
NETWORK
TITLE =

      A     M    507.7;
      A     M   1010.2;
      AN    Q    148.3;
      A     M   1050.2;
      AN    Q    268.3;
      A     M   1090.2;
      AN    Q    269.3;
      =     M    512.5;
NETWORK
TITLE =

      A     I     45.7;
      AN    I     48.0;
      AN    I     48.1;
      AN    I     48.2;
      A     I     65.0;
      AN    I     65.1;
      AN    I     65.2;
      AN    I     65.3;
      =     M    513.1;
NETWORK
TITLE =

      A     I     48.0;
      AN    I     45.7;
      AN    I     48.1;
      AN    I     48.2;
      A     I     65.1;
      AN    I     65.0;
      AN    I     65.2;
      AN    I     65.3;
      =     M    513.2;
NETWORK
TITLE =

      A     I     48.1;
      AN    I     45.7;
      AN    I     48.0;
      AN    I     48.2;
      A     I     65.2;
      AN    I     65.0;
      AN    I     65.1;
      AN    I     65.3;
      =     M    513.3;
NETWORK
TITLE =

      A     I     48.2;
      AN    I     45.7;
      AN    I     48.0;
      AN    I     48.1;
      A     I     65.3;
      AN    I     65.0;
      AN    I     65.1;
      AN    I     65.2;
      =     M    513.4;
NETWORK
TITLE =

      O     M    513.1;
      O     M    513.2;
      O     M    513.3;
      O     M    513.4;
      =     M    513.5;
NETWORK
TITLE =

      A(    ;
      A     M    500.6;
      A     M    502.2;
      A     M    501.0;
      A     M   4304.1;
      AN    M    510.0;
      A     M    513.1;
      AN    M   2010.0;
      O     ;
      A     M    500.5;
      A     DB51.DBX    1.0;
      A     DB51.DBX    3.6;
      AN    DB51.DBX    3.7;
      )     ;
      AN    M   2010.0;
      A     M    513.5;
      A     M    507.1;
      A     M    507.3;
      AN    M    507.6;
      =     Q     52.0;
NETWORK
TITLE =

      A(    ;
      A     M    500.6;
      AN    M    501.0;
      A     M    502.3;
      AN    M    510.1;
      AN    M    511.1;
      A     M    513.1;
      O     ;
      A     M    500.5;
      A     DB51.DBX    1.0;
      A     DB51.DBX    3.7;
      AN    DB51.DBX    3.6;
      )     ;
      A     M    513.5;
      A     M    507.3;
      AN    M    507.7;
      =     Q     52.1;
NETWORK
TITLE =
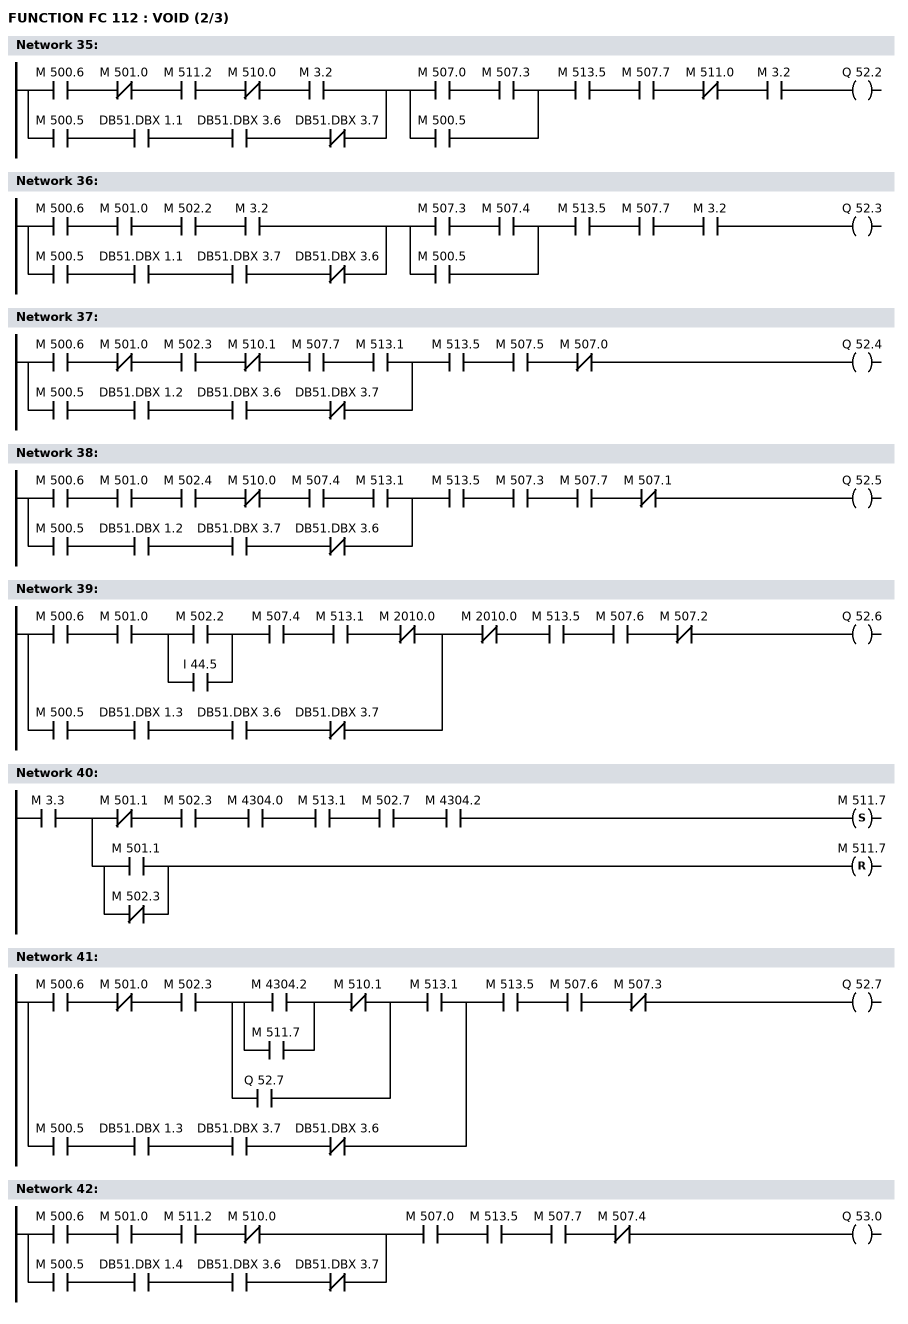

      A(    ;
      A     M    500.6;
      AN    M    501.0;
      A     M    511.2;
      AN    M    510.0;
      A     M      3.2;
      O     ;
      A     M    500.5;
      A     DB51.DBX    1.1;
      A     DB51.DBX    3.6;
      AN    DB51.DBX    3.7;
      )     ;
      A(    ;
      A     M    507.0;
      A     M    507.3;
      O     M    500.5;
      )     ;
      A     M    513.5;
      A     M    507.7;
      AN    M    511.0;
      A     M      3.2;
      =     Q     52.2;
NETWORK
TITLE =

      A(    ;
      A     M    500.6;
      A     M    501.0;
      A     M    502.2;
      A     M      3.2;
      O     ;
      A     M    500.5;
      A     DB51.DBX    1.1;
      A     DB51.DBX    3.7;
      AN    DB51.DBX    3.6;
      )     ;
      A(    ;
      A     M    507.3;
      A     M    507.4;
      O     M    500.5;
      )     ;
      A     M    513.5;
      A     M    507.7;
      A     M      3.2;
      =     Q     52.3;
NETWORK
TITLE =

      A(    ;
      A     M    500.6;
      AN    M    501.0;
      A     M    502.3;
      AN    M    510.1;
      A     M    507.7;
      A     M    513.1;
      O     ;
      A     M    500.5;
      A     DB51.DBX    1.2;
      A     DB51.DBX    3.6;
      AN    DB51.DBX    3.7;
      )     ;
      A     M    513.5;
      A     M    507.5;
      AN    M    507.0;
      =     Q     52.4;
NETWORK
TITLE =

      A(    ;
      A     M    500.6;
      A     M    501.0;
      A     M    502.4;
      AN    M    510.0;
      A     M    507.4;
      A     M    513.1;
      O     ;
      A     M    500.5;
      A     DB51.DBX    1.2;
      A     DB51.DBX    3.7;
      AN    DB51.DBX    3.6;
      )     ;
      A     M    513.5;
      A     M    507.3;
      A     M    507.7;
      AN    M    507.1;
      =     Q     52.5;
NETWORK
TITLE =

      A(    ;
      A     M    500.6;
      A     M    501.0;
      A(    ;
      O     M    502.2;
      O     I     44.5;
      )     ;
      A     M    507.4;
      A     M    513.1;
      AN    M   2010.0;
      O     ;
      A     M    500.5;
      A     DB51.DBX    1.3;
      A     DB51.DBX    3.6;
      AN    DB51.DBX    3.7;
      )     ;
      AN    M   2010.0;
      A     M    513.5;
      A     M    507.6;
      AN    M    507.2;
      =     Q     52.6;
NETWORK
TITLE =

      A     M      3.3;
      =     L      0.0;
      A     L      0.0;
      AN    M    501.1;
      A     M    502.3;
      A     M   4304.0;
      A     M    513.1;
      A     M    502.7;
      A     M   4304.2;
      S     M    511.7;
      A     L      0.0;
      A(    ;
      O     M    501.1;
      ON    M    502.3;
      )     ;
      R     M    511.7;
NETWORK
TITLE =

      A(    ;
      A     M    500.6;
      AN    M    501.0;
      A     M    502.3;
      A(    ;
      A(    ;
      O     M   4304.2;
      O     M    511.7;
      )     ;
      AN    M    510.1;
      O     Q     52.7;
      )     ;
      A     M    513.1;
      O     ;
      A     M    500.5;
      A     DB51.DBX    1.3;
      A     DB51.DBX    3.7;
      AN    DB51.DBX    3.6;
      )     ;
      A     M    513.5;
      A     M    507.6;
      AN    M    507.3;
      =     Q     52.7;
NETWORK
TITLE =

      A(    ;
      A     M    500.6;
      A     M    501.0;
      A     M    511.2;
      AN    M    510.0;
      O     ;
      A     M    500.5;
      A     DB51.DBX    1.4;
      A     DB51.DBX    3.6;
      AN    DB51.DBX    3.7;
      )     ;
      A     M    507.0;
      A     M    513.5;
      A     M    507.7;
      AN    M    507.4;
      =     Q     53.0;
NETWORK
TITLE =
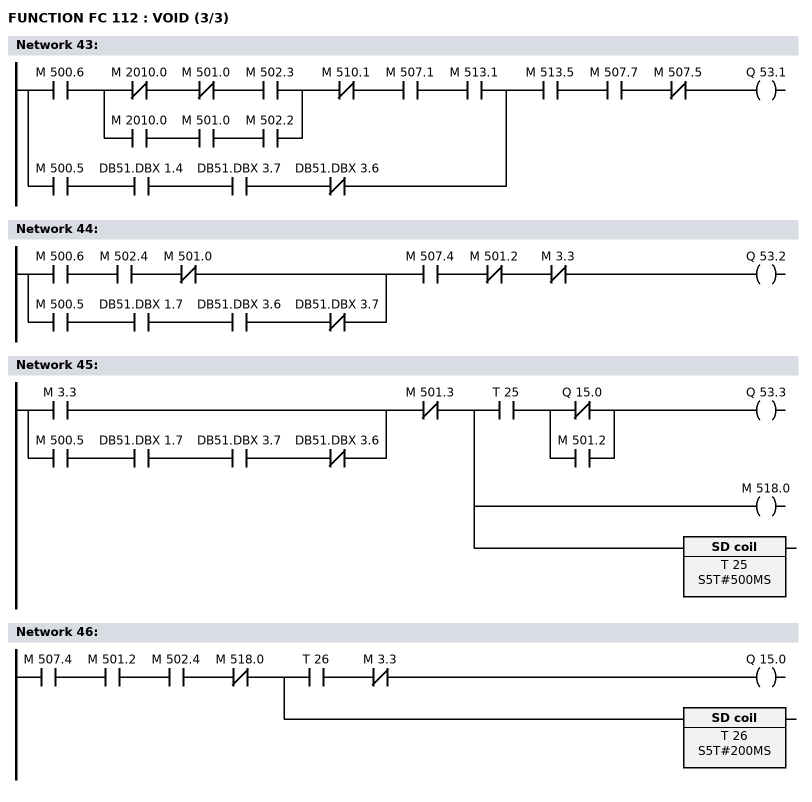

      A(    ;
      A     M    500.6;
      A(    ;
      AN    M   2010.0;
      AN    M    501.0;
      A     M    502.3;
      O     ;
      A     M   2010.0;
      A     M    501.0;
      A     M    502.2;
      )     ;
      AN    M    510.1;
      A     M    507.1;
      A     M    513.1;
      O     ;
      A     M    500.5;
      A     DB51.DBX    1.4;
      A     DB51.DBX    3.7;
      AN    DB51.DBX    3.6;
      )     ;
      A     M    513.5;
      A     M    507.7;
      AN    M    507.5;
      =     Q     53.1;
NETWORK
TITLE =

      A(    ;
      A     M    500.6;
      A     M    502.4;
      AN    M    501.0;
      O     ;
      A     M    500.5;
      A     DB51.DBX    1.7;
      A     DB51.DBX    3.6;
      AN    DB51.DBX    3.7;
      )     ;
      A     M    507.4;
      AN    M    501.2;
      AN    M      3.3;
      =     Q     53.2;
NETWORK
TITLE =

      A(    ;
      O     M      3.3;
      O     ;
      A     M    500.5;
      A     DB51.DBX    1.7;
      A     DB51.DBX    3.7;
      AN    DB51.DBX    3.6;
      )     ;
      AN    M    501.3;
      =     L      0.0;
      A     L      0.0;
      A     T     25;
      A(    ;
      ON    Q     15.0;
      O     M    501.2;
      )     ;
      =     Q     53.3;
      A     L      0.0;
      BLD   102;
      =     M    518.0;
      A     L      0.0;
      BLD   102;
      L     S5T#500MS;
      SD    T     25;
NETWORK
TITLE =

      A     M    507.4;
      A     M    501.2;
      A     M    502.4;
      AN    M    518.0;
      =     L      0.0;
      A     L      0.0;
      A     T     26;
      AN    M      3.3;
      =     Q     15.0;
      A     L      0.0;
      BLD   102;
      L     S5T#200MS;
      SD    T     26;
END_FUNCTION

FUNCTION FC 113 : VOID
TITLE =
VERSION : 0.1

BEGIN
NETWORK
TITLE =

      O     M    512.0;
      O     M    512.1;
      O     ;
      A     M    512.2;
      A     OV;
      O     M    512.3;
      =     Q     72.0;
NETWORK
TITLE =
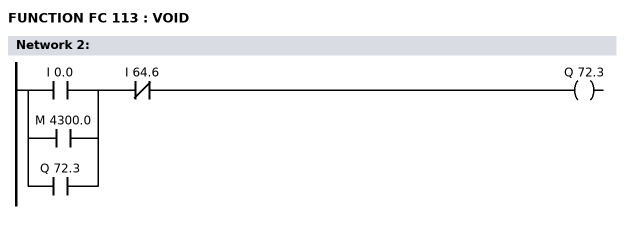

      A(    ;
      O     I      0.0;
      O     M   4300.0;
      O     Q     72.3;
      )     ;
      AN    I     64.6;
      =     Q     72.3;
NETWORK
TITLE =

      O     M    512.0;
      O     M    512.1;
      O     ;
      A     M    512.2;
      A     OV;
      O     M    512.3;
      =     L      0.0;
      A     L      0.0;
      A     T    201;
      AN    T    200;
      =     Q     72.4;
      A     L      0.0;
      BLD   102;
      L     S5T#2S;
      SD    T    200;
      A     L      0.0;
      BLD   102;
      L     S5T#500MS;
      SD    T    201;
NETWORK
TITLE =

      A     M    500.0;
      =     Q     72.5;
NETWORK
TITLE =

      A     Q     72.3;
      =     L      0.0;
      A     L      0.0;
      A(    ;
      A     M    500.5;
      A     DB51.DBX    3.0;
      O     M    512.3;
      )     ;
      =     Q     73.0;
      A     L      0.0;
      A(    ;
      A     M    500.5;
      A     DB51.DBX    3.1;
      O     M    512.0;
      )     ;
      =     Q     73.1;
      A     L      0.0;
      A(    ;
      A     M    500.5;
      A     DB51.DBX    3.2;
      O     M    512.1;
      )     ;
      =     Q     73.2;
      A     L      0.0;
      A     M    500.5;
      A     DB51.DBX    3.3;
      A     OV;
      =     Q     73.3;
NETWORK
TITLE =
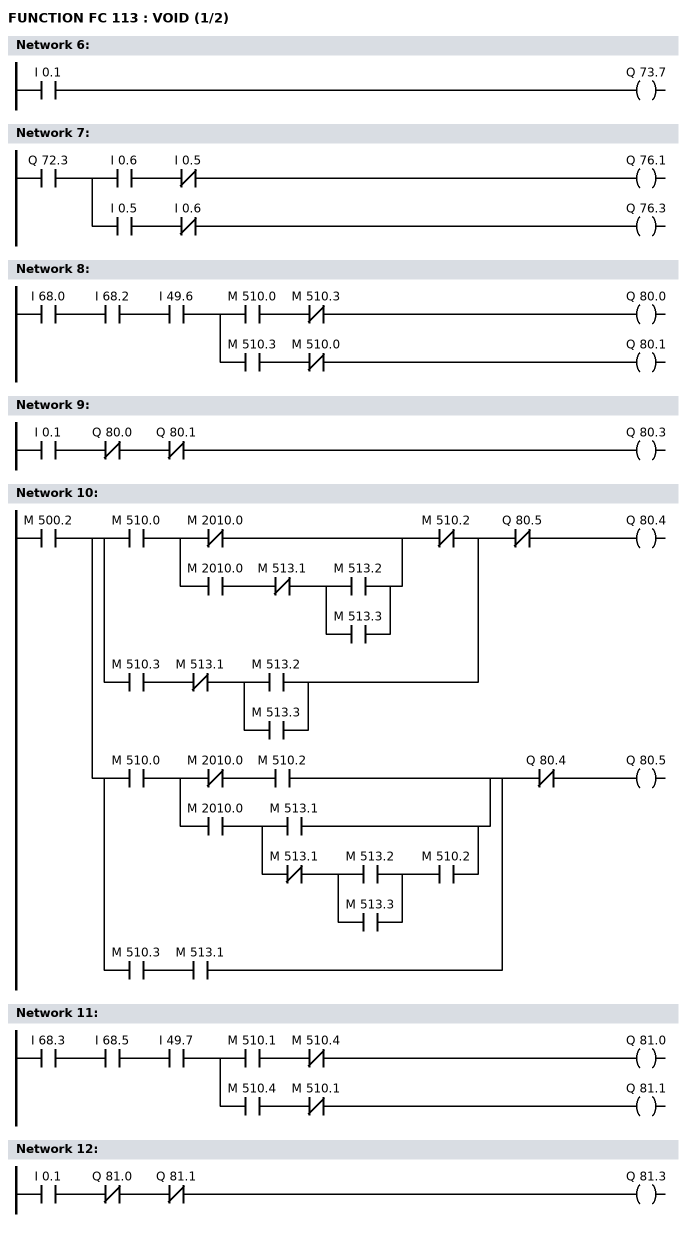

      A     I      0.1;
      =     Q     73.7;
NETWORK
TITLE =

      A     Q     72.3;
      =     L      0.0;
      A     L      0.0;
      A     I      0.6;
      AN    I      0.5;
      =     Q     76.1;
      A     L      0.0;
      A     I      0.5;
      AN    I      0.6;
      =     Q     76.3;
NETWORK
TITLE =

      A     I     68.0;
      A     I     68.2;
      A     I     49.6;
      =     L      0.0;
      A     L      0.0;
      A     M    510.0;
      AN    M    510.3;
      =     Q     80.0;
      A     L      0.0;
      A     M    510.3;
      AN    M    510.0;
      =     Q     80.1;
NETWORK
TITLE =

      A     I      0.1;
      AN    Q     80.0;
      AN    Q     80.1;
      =     Q     80.3;
NETWORK
TITLE =

      A     M    500.2;
      =     L      0.0;
      A     L      0.0;
      A(    ;
      A     M    510.0;
      A(    ;
      ON    M   2010.0;
      O     ;
      A     M   2010.0;
      AN    M    513.1;
      A(    ;
      O     M    513.2;
      O     M    513.3;
      )     ;
      )     ;
      AN    M    510.2;
      O     ;
      A     M    510.3;
      AN    M    513.1;
      A(    ;
      O     M    513.2;
      O     M    513.3;
      )     ;
      )     ;
      AN    Q     80.5;
      =     Q     80.4;
      A     L      0.0;
      A(    ;
      A     M    510.0;
      A(    ;
      AN    M   2010.0;
      A     M    510.2;
      O     ;
      A     M   2010.0;
      A(    ;
      O     M    513.1;
      O     ;
      AN    M    513.1;
      A(    ;
      O     M    513.2;
      O     M    513.3;
      )     ;
      A     M    510.2;
      )     ;
      )     ;
      O     ;
      A     M    510.3;
      A     M    513.1;
      )     ;
      AN    Q     80.4;
      =     Q     80.5;
NETWORK
TITLE =

      A     I     68.3;
      A     I     68.5;
      A     I     49.7;
      =     L      0.0;
      A     L      0.0;
      A     M    510.1;
      AN    M    510.4;
      =     Q     81.0;
      A     L      0.0;
      A     M    510.4;
      AN    M    510.1;
      =     Q     81.1;
NETWORK
TITLE =

      A     I      0.1;
      AN    Q     81.0;
      AN    Q     81.1;
      =     Q     81.3;
NETWORK
TITLE =
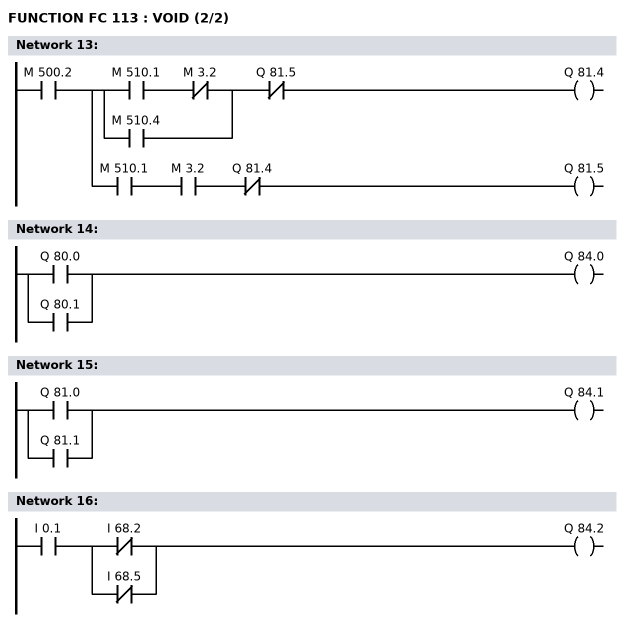

      A     M    500.2;
      =     L      0.0;
      A     L      0.0;
      A(    ;
      A     M    510.1;
      AN    M      3.2;
      O     M    510.4;
      )     ;
      AN    Q     81.5;
      =     Q     81.4;
      A     L      0.0;
      A     M    510.1;
      A     M      3.2;
      AN    Q     81.4;
      =     Q     81.5;
NETWORK
TITLE =

      O     Q     80.0;
      O     Q     80.1;
      =     Q     84.0;
NETWORK
TITLE =

      O     Q     81.0;
      O     Q     81.1;
      =     Q     84.1;
NETWORK
TITLE =

      A     I      0.1;
      A(    ;
      ON    I     68.2;
      ON    I     68.5;
      )     ;
      =     Q     84.2;
END_FUNCTION

FUNCTION_BLOCK FB 120
TITLE =
VERSION : 0.1


VAR
  S_RETURN_MODE : FB 402;
END_VAR
BEGIN
NETWORK
TITLE =
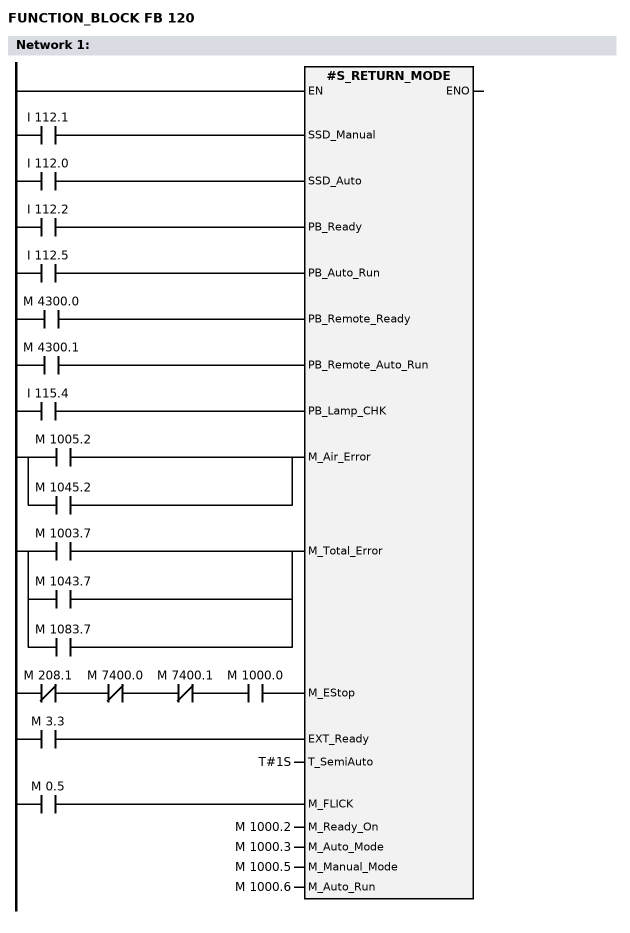

      A     I    112.1;
      =     L      0.0;
      BLD   103;
      A     I    112.0;
      =     L      0.1;
      BLD   103;
      A     I    112.2;
      =     L      0.2;
      BLD   103;
      A     I    112.5;
      =     L      0.3;
      BLD   103;
      A     M   4300.0;
      =     L      0.4;
      BLD   103;
      A     M   4300.1;
      =     L      0.5;
      BLD   103;
      A     I    115.4;
      =     L      0.6;
      BLD   103;
      A(    ;
      O     M   1005.2;
      O     M   1045.2;
      )     ;
      =     L      0.7;
      BLD   103;
      A(    ;
      O     M   1003.7;
      O     M   1043.7;
      O     M   1083.7;
      )     ;
      =     L      1.1;
      BLD   103;
      AN    M    208.1;
      AN    M   7400.0;
      AN    M   7400.1;
      A     M   1000.0;
      =     L      1.2;
      BLD   103;
      A     M      3.3;
      =     L      1.3;
      BLD   103;
      A     M      0.5;
      =     L      1.5;
      BLD   103;
      CALL #S_RETURN_MODE (
           SSD_Manual               := L      0.0,
           SSD_Auto                 := L      0.1,
           PB_Ready                 := L      0.2,
           PB_Auto_Run              := L      0.3,
           PB_Remote_Ready          := L      0.4,
           PB_Remote_Auto_Run       := L      0.5,
           PB_Lamp_CHK              := L      0.6,
           M_Air_Error              := L      0.7,
           M_Total_Error            := L      1.1,
           M_EStop                  := L      1.2,
           EXT_Ready                := L      1.3,
           T_SemiAuto               := T#1S,
           M_FLICK                  := L      1.5,
           M_Ready_On               := M   1000.2,
           M_Auto_Mode              := M   1000.3,
           M_Manual_Mode            := M   1000.5,
           M_Auto_Run               := M   1000.6);

      NOP   0;
END_FUNCTION_BLOCK

DATA_BLOCK DB 120
TITLE =
VERSION : 0.0

 FB 120
BEGIN
   S_RETURN_MODE.SSD_Manual := FALSE;
   S_RETURN_MODE.SSD_Auto := FALSE;
   S_RETURN_MODE.PB_Ready := FALSE;
   S_RETURN_MODE.PB_Auto_Run := FALSE;
   S_RETURN_MODE.PB_Remote_Ready := FALSE;
   S_RETURN_MODE.PB_Remote_Auto_Run := FALSE;
   S_RETURN_MODE.PB_Lamp_CHK := FALSE;
   S_RETURN_MODE.M_Air_Error := FALSE;
   S_RETURN_MODE.M_Water_Error := FALSE;
   S_RETURN_MODE.M_Total_Error := FALSE;
   S_RETURN_MODE.M_EStop := FALSE;
   S_RETURN_MODE.EXT_Ready := FALSE;
   S_RETURN_MODE.EXT_Auto := FALSE;
   S_RETURN_MODE.T_SemiAuto := T#0MS;
   S_RETURN_MODE.M_FLICK := FALSE;
   S_RETURN_MODE.M_Ready_On := FALSE;
   S_RETURN_MODE.M_Auto_Mode := FALSE;
   S_RETURN_MODE.M_SemiAuto_Mode := FALSE;
   S_RETURN_MODE.M_Manual_Mode := FALSE;
   S_RETURN_MODE.M_Auto_Run := FALSE;
   S_RETURN_MODE.LP_Ready_On := FALSE;
   S_RETURN_MODE.LP_Auto_Run := FALSE;
   S_RETURN_MODE.AUTO_MODE_DELAY.IN := FALSE;
   S_RETURN_MODE.AUTO_MODE_DELAY.PT := T#0MS;
   S_RETURN_MODE.AUTO_MODE_DELAY.Q := FALSE;
   S_RETURN_MODE.AUTO_MODE_DELAY.ET := T#0MS;
   S_RETURN_MODE.AUTO_MODE_DELAY.STATE := B#16#0;
   S_RETURN_MODE.AUTO_MODE_DELAY.STIME := T#0MS;
   S_RETURN_MODE.AUTO_MODE_DELAY.ATIME := T#0MS;
   S_RETURN_MODE.SEMI_AUTO_DELAY.IN := FALSE;
   S_RETURN_MODE.SEMI_AUTO_DELAY.PT := T#0MS;
   S_RETURN_MODE.SEMI_AUTO_DELAY.Q := FALSE;
   S_RETURN_MODE.SEMI_AUTO_DELAY.ET := T#0MS;
   S_RETURN_MODE.SEMI_AUTO_DELAY.STATE := B#16#0;
   S_RETURN_MODE.SEMI_AUTO_DELAY.STIME := T#0MS;
   S_RETURN_MODE.SEMI_AUTO_DELAY.ATIME := T#0MS;
   S_RETURN_MODE.MANUAL_DELAY.IN := FALSE;
   S_RETURN_MODE.MANUAL_DELAY.PT := T#0MS;
   S_RETURN_MODE.MANUAL_DELAY.Q := FALSE;
   S_RETURN_MODE.MANUAL_DELAY.ET := T#0MS;
   S_RETURN_MODE.MANUAL_DELAY.STATE := B#16#0;
   S_RETURN_MODE.MANUAL_DELAY.STIME := T#0MS;
   S_RETURN_MODE.MANUAL_DELAY.ATIME := T#0MS;
END_DATA_BLOCK

FUNCTION FC 120 : VOID
TITLE =
VERSION : 0.1

BEGIN
NETWORK
TITLE =
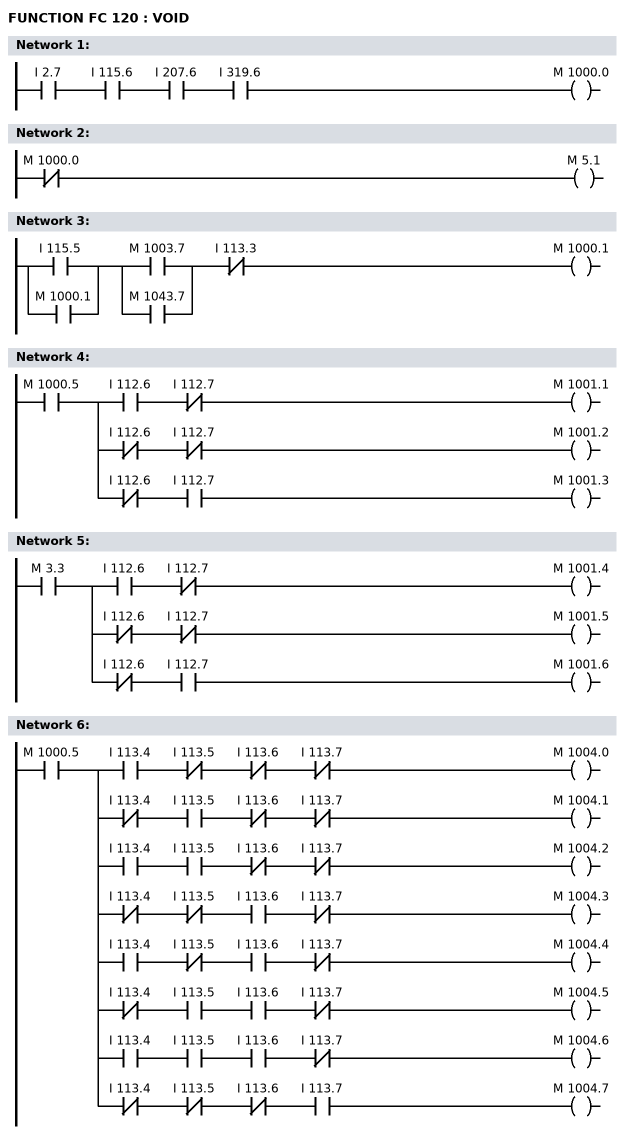

      A     I      2.7;
      A     I    115.6;
      A     I    207.6;
      A     I    319.6;
      =     M   1000.0;
NETWORK
TITLE =

      AN    M   1000.0;
      =     M      5.1;
NETWORK
TITLE =

      A(    ;
      O     I    115.5;
      O     M   1000.1;
      )     ;
      A(    ;
      O     M   1003.7;
      O     M   1043.7;
      )     ;
      AN    I    113.3;
      =     M   1000.1;
NETWORK
TITLE =

      A     M   1000.5;
      =     L      0.0;
      A     L      0.0;
      A     I    112.6;
      AN    I    112.7;
      =     M   1001.1;
      A     L      0.0;
      AN    I    112.6;
      AN    I    112.7;
      =     M   1001.2;
      A     L      0.0;
      AN    I    112.6;
      A     I    112.7;
      =     M   1001.3;
NETWORK
TITLE =

      A     M      3.3;
      =     L      0.0;
      A     L      0.0;
      A     I    112.6;
      AN    I    112.7;
      =     M   1001.4;
      A     L      0.0;
      AN    I    112.6;
      AN    I    112.7;
      =     M   1001.5;
      A     L      0.0;
      AN    I    112.6;
      A     I    112.7;
      =     M   1001.6;
NETWORK
TITLE =

      A     M   1000.5;
      =     L      0.0;
      A     L      0.0;
      A     I    113.4;
      AN    I    113.5;
      AN    I    113.6;
      AN    I    113.7;
      =     M   1004.0;
      A     L      0.0;
      AN    I    113.4;
      A     I    113.5;
      AN    I    113.6;
      AN    I    113.7;
      =     M   1004.1;
      A     L      0.0;
      A     I    113.4;
      A     I    113.5;
      AN    I    113.6;
      AN    I    113.7;
      =     M   1004.2;
      A     L      0.0;
      AN    I    113.4;
      AN    I    113.5;
      A     I    113.6;
      AN    I    113.7;
      =     M   1004.3;
      A     L      0.0;
      A     I    113.4;
      AN    I    113.5;
      A     I    113.6;
      AN    I    113.7;
      =     M   1004.4;
      A     L      0.0;
      AN    I    113.4;
      A     I    113.5;
      A     I    113.6;
      AN    I    113.7;
      =     M   1004.5;
      A     L      0.0;
      A     I    113.4;
      A     I    113.5;
      A     I    113.6;
      AN    I    113.7;
      =     M   1004.6;
      A     L      0.0;
      AN    I    113.4;
      AN    I    113.5;
      AN    I    113.6;
      A     I    113.7;
      =     M   1004.7;
END_FUNCTION

FUNCTION_BLOCK FB 121
TITLE =
VERSION : 0.1


VAR
  S_RTN1_STP1 : FB 424;
  S_RTN1_STP2 : FB 424;
  S_RTN1_STP3 : FB 424;
  S_RTN1_STP4 : FB 424;
  S_RTN2_STP1 : FB 424;
  S_RTN2_STP2 : FB 424;
  S_RTN3_STP1 : FB 424;
  S_RTN3_STP2 : FB 424;
END_VAR
BEGIN
NETWORK
TITLE =RETURN1 L/S이상

NETWORK
TITLE =
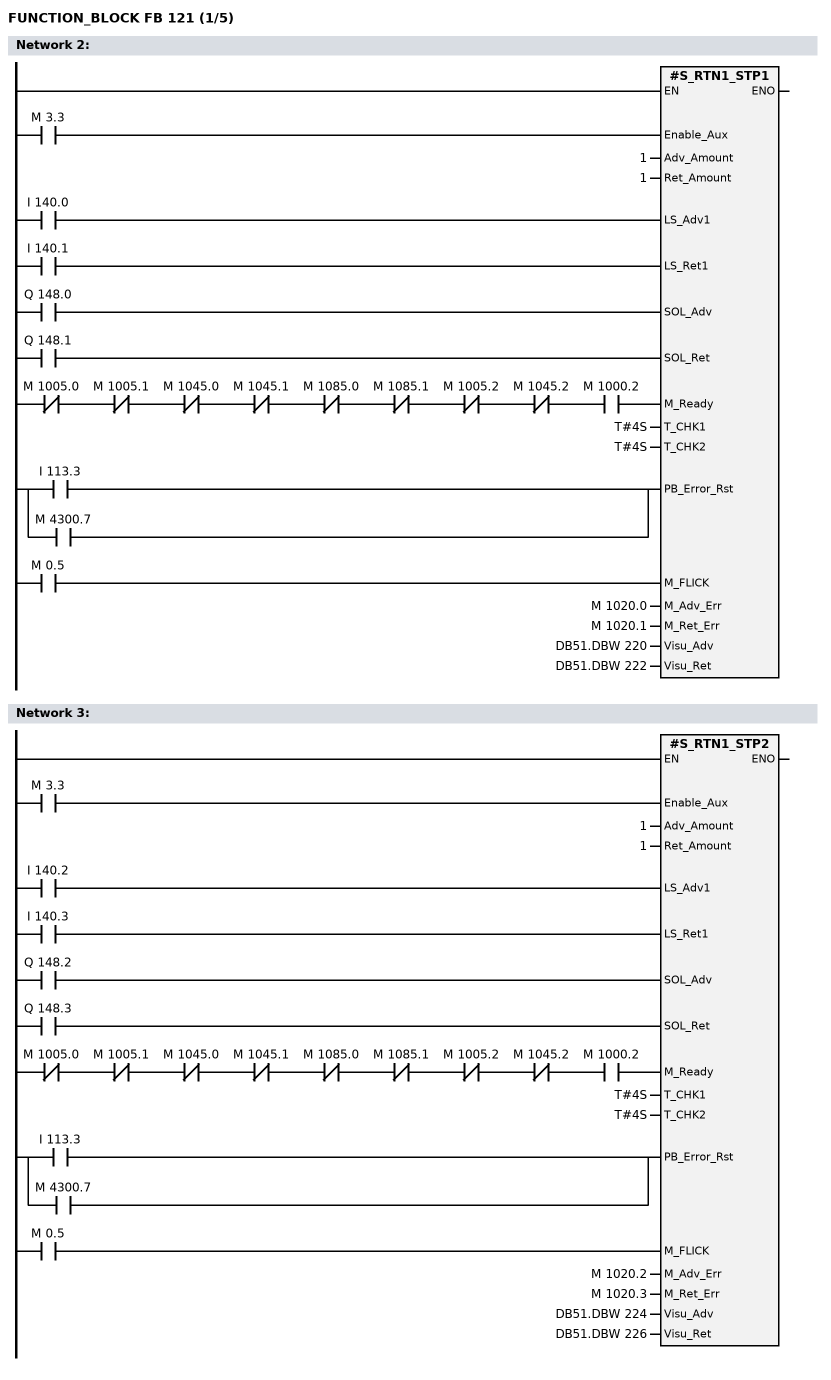

      A     M      3.3;
      =     L      0.0;
      BLD   103;
      A     I    140.0;
      =     L      0.1;
      BLD   103;
      A     I    140.1;
      =     L      0.2;
      BLD   103;
      A     Q    148.0;
      =     L      1.1;
      BLD   103;
      A     Q    148.1;
      =     L      1.2;
      BLD   103;
      AN    M   1005.0;
      AN    M   1005.1;
      AN    M   1045.0;
      AN    M   1045.1;
      AN    M   1085.0;
      AN    M   1085.1;
      AN    M   1005.2;
      AN    M   1045.2;
      A     M   1000.2;
      =     L      1.3;
      BLD   103;
      A(    ;
      O     I    113.3;
      O     M   4300.7;
      )     ;
      =     L      1.5;
      BLD   103;
      A     M      0.5;
      =     L      1.6;
      BLD   103;
      CALL #S_RTN1_STP1 (
           Enable_Aux               := L      0.0,
           Adv_Amount               := 1,
           Ret_Amount               := 1,
           LS_Adv1                  := L      0.1,
           LS_Ret1                  := L      0.2,
           SOL_Adv                  := L      1.1,
           SOL_Ret                  := L      1.2,
           M_Ready                  := L      1.3,
           T_CHK1                   := T#4S,
           T_CHK2                   := T#4S,
           PB_Error_Rst             := L      1.5,
           M_FLICK                  := L      1.6,
           M_Adv_Err                := M   1020.0,
           M_Ret_Err                := M   1020.1,
           Visu_Adv                 := DB51.DBW  220,
           Visu_Ret                 := DB51.DBW  222);
      NOP   0;
NETWORK
TITLE =

      A     M      3.3;
      =     L      0.0;
      BLD   103;
      A     I    140.2;
      =     L      0.1;
      BLD   103;
      A     I    140.3;
      =     L      0.2;
      BLD   103;
      A     Q    148.2;
      =     L      1.1;
      BLD   103;
      A     Q    148.3;
      =     L      1.2;
      BLD   103;
      AN    M   1005.0;
      AN    M   1005.1;
      AN    M   1045.0;
      AN    M   1045.1;
      AN    M   1085.0;
      AN    M   1085.1;
      AN    M   1005.2;
      AN    M   1045.2;
      A     M   1000.2;
      =     L      1.3;
      BLD   103;
      A(    ;
      O     I    113.3;
      O     M   4300.7;
      )     ;
      =     L      1.5;
      BLD   103;
      A     M      0.5;
      =     L      1.6;
      BLD   103;
      CALL #S_RTN1_STP2 (
           Enable_Aux               := L      0.0,
           Adv_Amount               := 1,
           Ret_Amount               := 1,
           LS_Adv1                  := L      0.1,
           LS_Ret1                  := L      0.2,
           SOL_Adv                  := L      1.1,
           SOL_Ret                  := L      1.2,
           M_Ready                  := L      1.3,
           T_CHK1                   := T#4S,
           T_CHK2                   := T#4S,
           PB_Error_Rst             := L      1.5,
           M_FLICK                  := L      1.6,
           M_Adv_Err                := M   1020.2,
           M_Ret_Err                := M   1020.3,
           Visu_Adv                 := DB51.DBW  224,
           Visu_Ret                 := DB51.DBW  226);
      NOP   0;
NETWORK
TITLE =
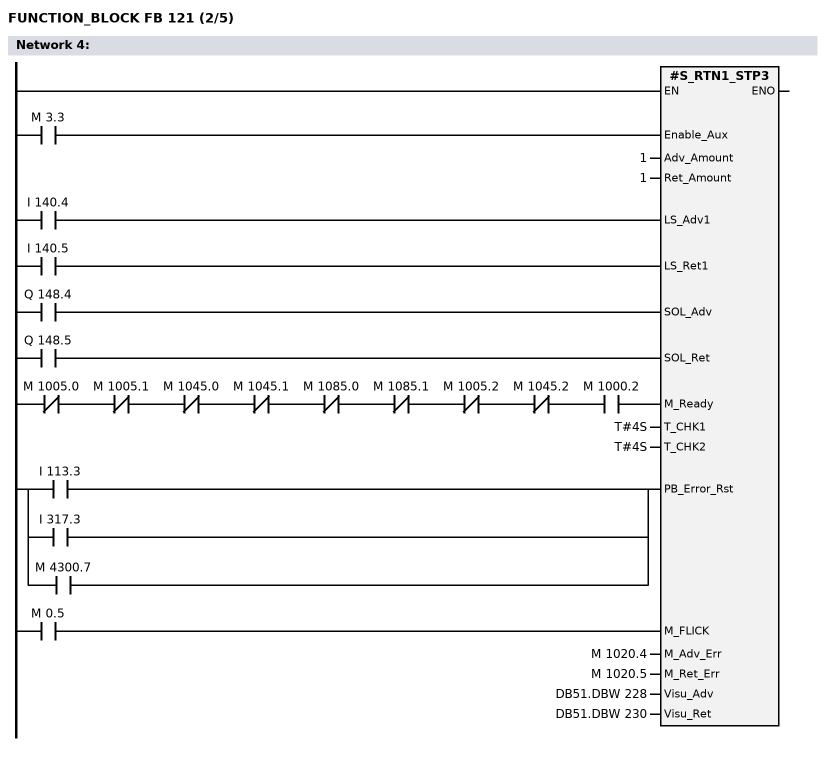

      A     M      3.3;
      =     L      0.0;
      BLD   103;
      A     I    140.4;
      =     L      0.1;
      BLD   103;
      A     I    140.5;
      =     L      0.2;
      BLD   103;
      A     Q    148.4;
      =     L      1.1;
      BLD   103;
      A     Q    148.5;
      =     L      1.2;
      BLD   103;
      AN    M   1005.0;
      AN    M   1005.1;
      AN    M   1045.0;
      AN    M   1045.1;
      AN    M   1085.0;
      AN    M   1085.1;
      AN    M   1005.2;
      AN    M   1045.2;
      A     M   1000.2;
      =     L      1.3;
      BLD   103;
      A(    ;
      O     I    113.3;
      O     I    317.3;
      O     M   4300.7;
      )     ;
      =     L      1.5;
      BLD   103;
      A     M      0.5;
      =     L      1.6;
      BLD   103;
      CALL #S_RTN1_STP3 (
           Enable_Aux               := L      0.0,
           Adv_Amount               := 1,
           Ret_Amount               := 1,
           LS_Adv1                  := L      0.1,
           LS_Ret1                  := L      0.2,
           SOL_Adv                  := L      1.1,
           SOL_Ret                  := L      1.2,
           M_Ready                  := L      1.3,
           T_CHK1                   := T#4S,
           T_CHK2                   := T#4S,
           PB_Error_Rst             := L      1.5,
           M_FLICK                  := L      1.6,
           M_Adv_Err                := M   1020.4,
           M_Ret_Err                := M   1020.5,
           Visu_Adv                 := DB51.DBW  228,
           Visu_Ret                 := DB51.DBW  230);
      NOP   0;
NETWORK
TITLE =
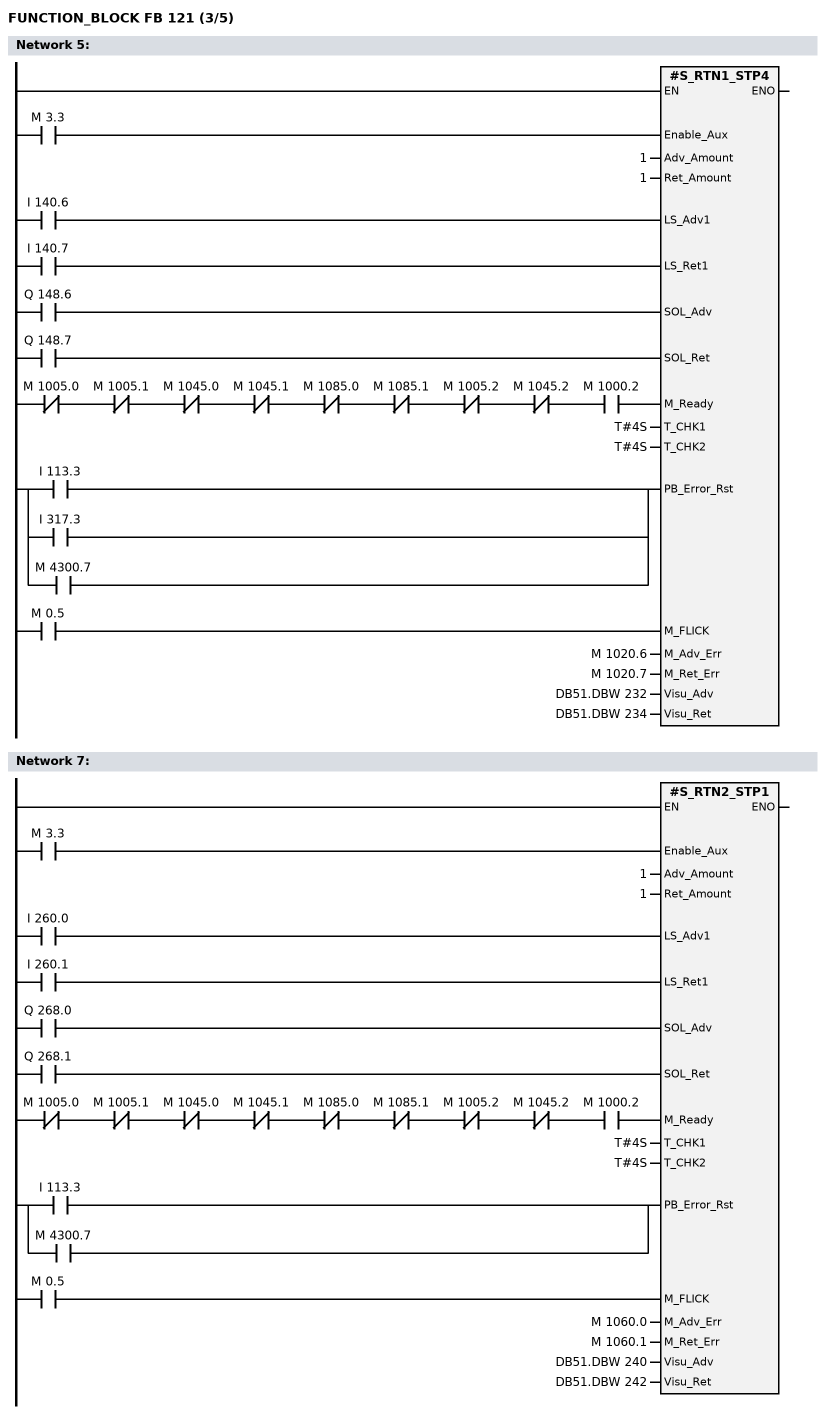

      A     M      3.3;
      =     L      0.0;
      BLD   103;
      A     I    140.6;
      =     L      0.1;
      BLD   103;
      A     I    140.7;
      =     L      0.2;
      BLD   103;
      A     Q    148.6;
      =     L      1.1;
      BLD   103;
      A     Q    148.7;
      =     L      1.2;
      BLD   103;
      AN    M   1005.0;
      AN    M   1005.1;
      AN    M   1045.0;
      AN    M   1045.1;
      AN    M   1085.0;
      AN    M   1085.1;
      AN    M   1005.2;
      AN    M   1045.2;
      A     M   1000.2;
      =     L      1.3;
      BLD   103;
      A(    ;
      O     I    113.3;
      O     I    317.3;
      O     M   4300.7;
      )     ;
      =     L      1.5;
      BLD   103;
      A     M      0.5;
      =     L      1.6;
      BLD   103;
      CALL #S_RTN1_STP4 (
           Enable_Aux               := L      0.0,
           Adv_Amount               := 1,
           Ret_Amount               := 1,
           LS_Adv1                  := L      0.1,
           LS_Ret1                  := L      0.2,
           SOL_Adv                  := L      1.1,
           SOL_Ret                  := L      1.2,
           M_Ready                  := L      1.3,
           T_CHK1                   := T#4S,
           T_CHK2                   := T#4S,
           PB_Error_Rst             := L      1.5,
           M_FLICK                  := L      1.6,
           M_Adv_Err                := M   1020.6,
           M_Ret_Err                := M   1020.7,
           Visu_Adv                 := DB51.DBW  232,
           Visu_Ret                 := DB51.DBW  234);
      NOP   0;
NETWORK
TITLE =RETURN2 L/S이상

NETWORK
TITLE =

      A     M      3.3;
      =     L      0.0;
      BLD   103;
      A     I    260.0;
      =     L      0.1;
      BLD   103;
      A     I    260.1;
      =     L      0.2;
      BLD   103;
      A     Q    268.0;
      =     L      1.1;
      BLD   103;
      A     Q    268.1;
      =     L      1.2;
      BLD   103;
      AN    M   1005.0;
      AN    M   1005.1;
      AN    M   1045.0;
      AN    M   1045.1;
      AN    M   1085.0;
      AN    M   1085.1;
      AN    M   1005.2;
      AN    M   1045.2;
      A     M   1000.2;
      =     L      1.3;
      BLD   103;
      A(    ;
      O     I    113.3;
      O     M   4300.7;
      )     ;
      =     L      1.5;
      BLD   103;
      A     M      0.5;
      =     L      1.6;
      BLD   103;
      CALL #S_RTN2_STP1 (
           Enable_Aux               := L      0.0,
           Adv_Amount               := 1,
           Ret_Amount               := 1,
           LS_Adv1                  := L      0.1,
           LS_Ret1                  := L      0.2,
           SOL_Adv                  := L      1.1,
           SOL_Ret                  := L      1.2,
           M_Ready                  := L      1.3,
           T_CHK1                   := T#4S,
           T_CHK2                   := T#4S,
           PB_Error_Rst             := L      1.5,
           M_FLICK                  := L      1.6,
           M_Adv_Err                := M   1060.0,
           M_Ret_Err                := M   1060.1,
           Visu_Adv                 := DB51.DBW  240,
           Visu_Ret                 := DB51.DBW  242);
      NOP   0;
NETWORK
TITLE =
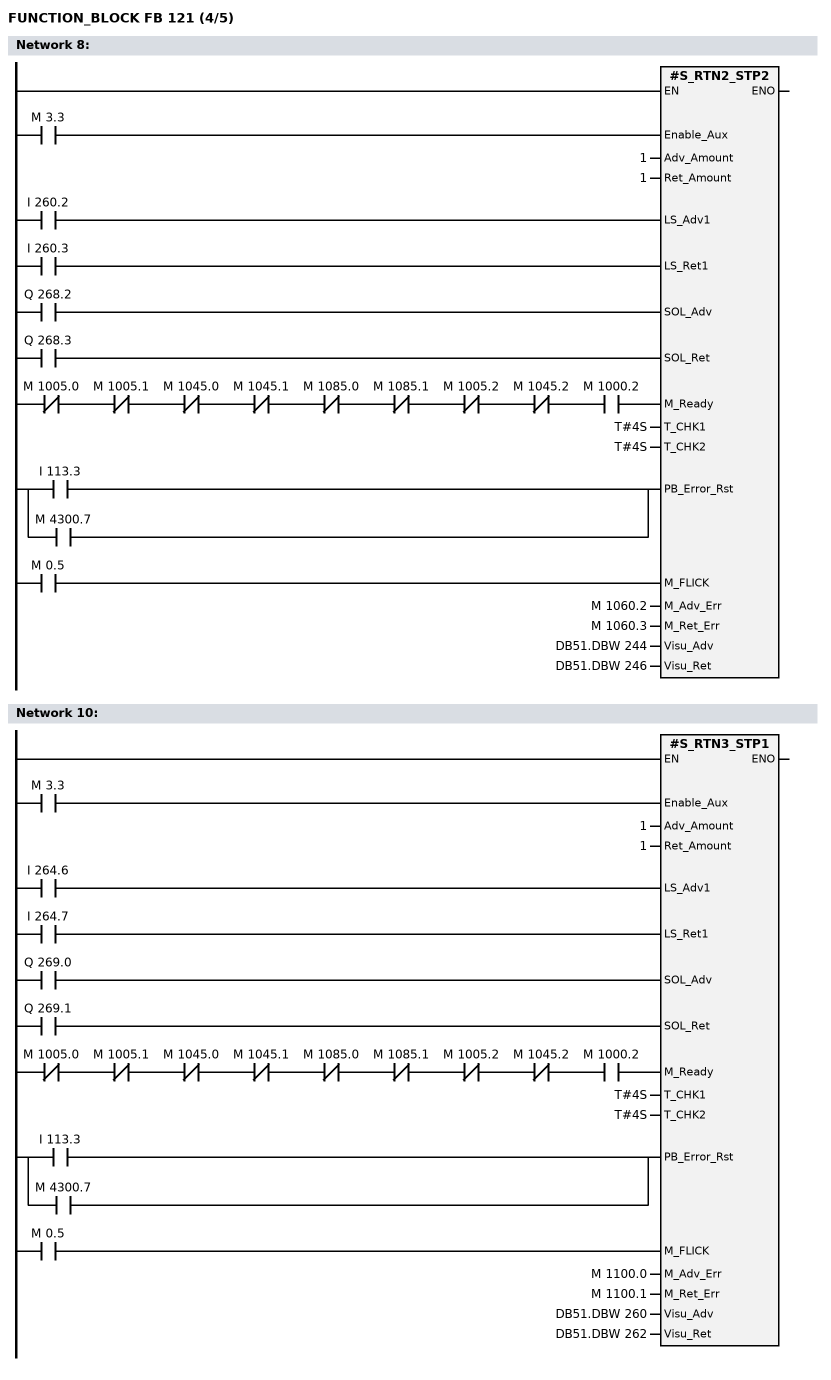

      A     M      3.3;
      =     L      0.0;
      BLD   103;
      A     I    260.2;
      =     L      0.1;
      BLD   103;
      A     I    260.3;
      =     L      0.2;
      BLD   103;
      A     Q    268.2;
      =     L      1.1;
      BLD   103;
      A     Q    268.3;
      =     L      1.2;
      BLD   103;
      AN    M   1005.0;
      AN    M   1005.1;
      AN    M   1045.0;
      AN    M   1045.1;
      AN    M   1085.0;
      AN    M   1085.1;
      AN    M   1005.2;
      AN    M   1045.2;
      A     M   1000.2;
      =     L      1.3;
      BLD   103;
      A(    ;
      O     I    113.3;
      O     M   4300.7;
      )     ;
      =     L      1.5;
      BLD   103;
      A     M      0.5;
      =     L      1.6;
      BLD   103;
      CALL #S_RTN2_STP2 (
           Enable_Aux               := L      0.0,
           Adv_Amount               := 1,
           Ret_Amount               := 1,
           LS_Adv1                  := L      0.1,
           LS_Ret1                  := L      0.2,
           SOL_Adv                  := L      1.1,
           SOL_Ret                  := L      1.2,
           M_Ready                  := L      1.3,
           T_CHK1                   := T#4S,
           T_CHK2                   := T#4S,
           PB_Error_Rst             := L      1.5,
           M_FLICK                  := L      1.6,
           M_Adv_Err                := M   1060.2,
           M_Ret_Err                := M   1060.3,
           Visu_Adv                 := DB51.DBW  244,
           Visu_Ret                 := DB51.DBW  246);
      NOP   0;
NETWORK
TITLE =RETURN3 L/S이상

NETWORK
TITLE =

      A     M      3.3;
      =     L      0.0;
      BLD   103;
      A     I    264.6;
      =     L      0.1;
      BLD   103;
      A     I    264.7;
      =     L      0.2;
      BLD   103;
      A     Q    269.0;
      =     L      1.1;
      BLD   103;
      A     Q    269.1;
      =     L      1.2;
      BLD   103;
      AN    M   1005.0;
      AN    M   1005.1;
      AN    M   1045.0;
      AN    M   1045.1;
      AN    M   1085.0;
      AN    M   1085.1;
      AN    M   1005.2;
      AN    M   1045.2;
      A     M   1000.2;
      =     L      1.3;
      BLD   103;
      A(    ;
      O     I    113.3;
      O     M   4300.7;
      )     ;
      =     L      1.5;
      BLD   103;
      A     M      0.5;
      =     L      1.6;
      BLD   103;
      CALL #S_RTN3_STP1 (
           Enable_Aux               := L      0.0,
           Adv_Amount               := 1,
           Ret_Amount               := 1,
           LS_Adv1                  := L      0.1,
           LS_Ret1                  := L      0.2,
           SOL_Adv                  := L      1.1,
           SOL_Ret                  := L      1.2,
           M_Ready                  := L      1.3,
           T_CHK1                   := T#4S,
           T_CHK2                   := T#4S,
           PB_Error_Rst             := L      1.5,
           M_FLICK                  := L      1.6,
           M_Adv_Err                := M   1100.0,
           M_Ret_Err                := M   1100.1,
           Visu_Adv                 := DB51.DBW  260,
           Visu_Ret                 := DB51.DBW  262);
      NOP   0;
NETWORK
TITLE =
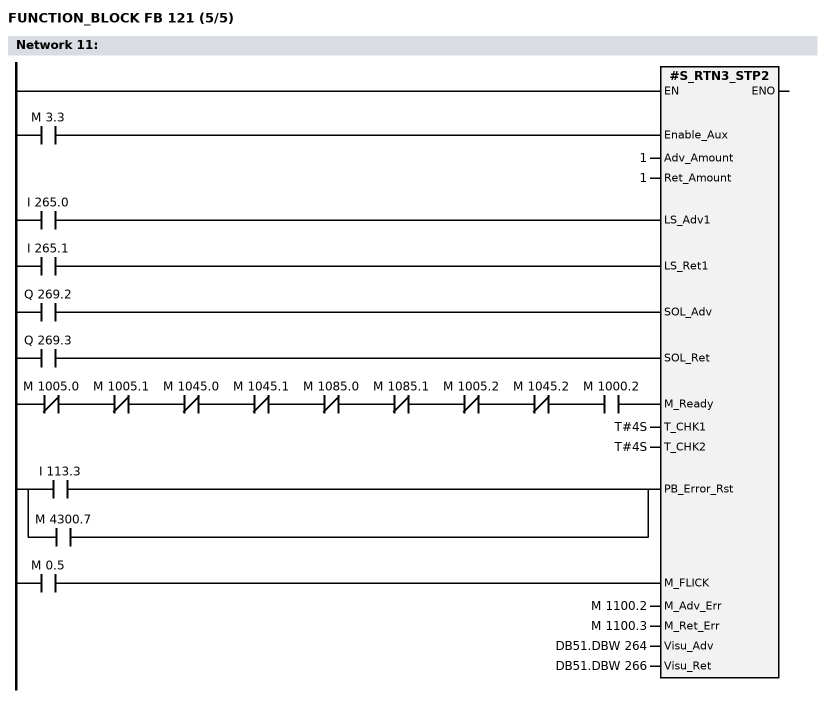

      A     M      3.3;
      =     L      0.0;
      BLD   103;
      A     I    265.0;
      =     L      0.1;
      BLD   103;
      A     I    265.1;
      =     L      0.2;
      BLD   103;
      A     Q    269.2;
      =     L      1.1;
      BLD   103;
      A     Q    269.3;
      =     L      1.2;
      BLD   103;
      AN    M   1005.0;
      AN    M   1005.1;
      AN    M   1045.0;
      AN    M   1045.1;
      AN    M   1085.0;
      AN    M   1085.1;
      AN    M   1005.2;
      AN    M   1045.2;
      A     M   1000.2;
      =     L      1.3;
      BLD   103;
      A(    ;
      O     I    113.3;
      O     M   4300.7;
      )     ;
      =     L      1.5;
      BLD   103;
      A     M      0.5;
      =     L      1.6;
      BLD   103;
      CALL #S_RTN3_STP2 (
           Enable_Aux               := L      0.0,
           Adv_Amount               := 1,
           Ret_Amount               := 1,
           LS_Adv1                  := L      0.1,
           LS_Ret1                  := L      0.2,
           SOL_Adv                  := L      1.1,
           SOL_Ret                  := L      1.2,
           M_Ready                  := L      1.3,
           T_CHK1                   := T#4S,
           T_CHK2                   := T#4S,
           PB_Error_Rst             := L      1.5,
           M_FLICK                  := L      1.6,
           M_Adv_Err                := M   1100.2,
           M_Ret_Err                := M   1100.3,
           Visu_Adv                 := DB51.DBW  264,
           Visu_Ret                 := DB51.DBW  266);
      NOP   0;
END_FUNCTION_BLOCK

DATA_BLOCK DB 121
TITLE =
VERSION : 0.0

 FB 121
BEGIN
   S_RTN1_STP1.Enable_Aux := FALSE;
   S_RTN1_STP1.Adv_Amount := 0;
   S_RTN1_STP1.Ret_Amount := 0;
   S_RTN1_STP1.LS_Adv1 := FALSE;
   S_RTN1_STP1.LS_Ret1 := FALSE;
   S_RTN1_STP1.LS_Adv2 := FALSE;
   S_RTN1_STP1.LS_Ret2 := FALSE;
   S_RTN1_STP1.LS_Adv3 := FALSE;
   S_RTN1_STP1.LS_Ret3 := FALSE;
   S_RTN1_STP1.LS_Adv4 := FALSE;
   S_RTN1_STP1.LS_Ret4 := FALSE;
   S_RTN1_STP1.SOL_Adv := FALSE;
   S_RTN1_STP1.SOL_Ret := FALSE;
   S_RTN1_STP1.M_Ready := FALSE;
   S_RTN1_STP1.T_CHK1 := T#0MS;
   S_RTN1_STP1.T_CHK2 := T#0MS;
   S_RTN1_STP1.PB_Lamp_CHK := FALSE;
   S_RTN1_STP1.PB_Error_Rst := FALSE;
   S_RTN1_STP1.M_FLICK := FALSE;
   S_RTN1_STP1.M_Adv_Err := FALSE;
   S_RTN1_STP1.M_Ret_Err := FALSE;
   S_RTN1_STP1.LP_Adv := FALSE;
   S_RTN1_STP1.LP_Ret := FALSE;
   S_RTN1_STP1.Visu_Adv := W#16#0;
   S_RTN1_STP1.Visu_Ret := W#16#0;
   S_RTN1_STP1.Error_T1.IN := FALSE;
   S_RTN1_STP1.Error_T1.PT := T#0MS;
   S_RTN1_STP1.Error_T1.Q := FALSE;
   S_RTN1_STP1.Error_T1.ET := T#0MS;
   S_RTN1_STP1.Error_T1.STATE := B#16#0;
   S_RTN1_STP1.Error_T1.STIME := T#0MS;
   S_RTN1_STP1.Error_T1.ATIME := T#0MS;
   S_RTN1_STP1.Error_T2.IN := FALSE;
   S_RTN1_STP1.Error_T2.PT := T#0MS;
   S_RTN1_STP1.Error_T2.Q := FALSE;
   S_RTN1_STP1.Error_T2.ET := T#0MS;
   S_RTN1_STP1.Error_T2.STATE := B#16#0;
   S_RTN1_STP1.Error_T2.STIME := T#0MS;
   S_RTN1_STP1.Error_T2.ATIME := T#0MS;
   S_RTN1_STP1.CHK_Aux1 := FALSE;
   S_RTN1_STP1.CHK_Aux2 := FALSE;
   S_RTN1_STP1.Error_T1_DN := FALSE;
   S_RTN1_STP1.Error_T2_DN := FALSE;
   S_RTN1_STP1.Adv_Memo := FALSE;
   S_RTN1_STP1.Visu_Adv_Arr[0] := FALSE;
   S_RTN1_STP1.Visu_Adv_Arr[1] := FALSE;
   S_RTN1_STP1.Visu_Adv_Arr[2] := FALSE;
   S_RTN1_STP1.Visu_Adv_Arr[3] := FALSE;
   S_RTN1_STP1.Visu_Adv_Arr[4] := FALSE;
   S_RTN1_STP1.Visu_Adv_Arr[5] := FALSE;
   S_RTN1_STP1.Visu_Adv_Arr[6] := FALSE;
   S_RTN1_STP1.Visu_Adv_Arr[7] := FALSE;
   S_RTN1_STP1.Visu_Adv_Arr[8] := FALSE;
   S_RTN1_STP1.Visu_Adv_Arr[9] := FALSE;
   S_RTN1_STP1.Visu_Adv_Arr[10] := FALSE;
   S_RTN1_STP1.Visu_Adv_Arr[11] := FALSE;
   S_RTN1_STP1.Visu_Adv_Arr[12] := FALSE;
   S_RTN1_STP1.Visu_Adv_Arr[13] := FALSE;
   S_RTN1_STP1.Visu_Adv_Arr[14] := FALSE;
   S_RTN1_STP1.Visu_Adv_Arr[15] := FALSE;
   S_RTN1_STP1.Visu_Ret_Arr[0] := FALSE;
   S_RTN1_STP1.Visu_Ret_Arr[1] := FALSE;
   S_RTN1_STP1.Visu_Ret_Arr[2] := FALSE;
   S_RTN1_STP1.Visu_Ret_Arr[3] := FALSE;
   S_RTN1_STP1.Visu_Ret_Arr[4] := FALSE;
   S_RTN1_STP1.Visu_Ret_Arr[5] := FALSE;
   S_RTN1_STP1.Visu_Ret_Arr[6] := FALSE;
   S_RTN1_STP1.Visu_Ret_Arr[7] := FALSE;
   S_RTN1_STP1.Visu_Ret_Arr[8] := FALSE;
   S_RTN1_STP1.Visu_Ret_Arr[9] := FALSE;
   S_RTN1_STP1.Visu_Ret_Arr[10] := FALSE;
   S_RTN1_STP1.Visu_Ret_Arr[11] := FALSE;
   S_RTN1_STP1.Visu_Ret_Arr[12] := FALSE;
   S_RTN1_STP1.Visu_Ret_Arr[13] := FALSE;
   S_RTN1_STP1.Visu_Ret_Arr[14] := FALSE;
   S_RTN1_STP1.Visu_Ret_Arr[15] := FALSE;
   S_RTN1_STP1.BLK_Move_Ret := 0;
   S_RTN1_STP1.Enable := FALSE;
   S_RTN1_STP1.Adv_End := FALSE;
   S_RTN1_STP1.Ret_End := FALSE;
   S_RTN1_STP2.Enable_Aux := FALSE;
   S_RTN1_STP2.Adv_Amount := 0;
   S_RTN1_STP2.Ret_Amount := 0;
   S_RTN1_STP2.LS_Adv1 := FALSE;
   S_RTN1_STP2.LS_Ret1 := FALSE;
   S_RTN1_STP2.LS_Adv2 := FALSE;
   S_RTN1_STP2.LS_Ret2 := FALSE;
   S_RTN1_STP2.LS_Adv3 := FALSE;
   S_RTN1_STP2.LS_Ret3 := FALSE;
   S_RTN1_STP2.LS_Adv4 := FALSE;
   S_RTN1_STP2.LS_Ret4 := FALSE;
   S_RTN1_STP2.SOL_Adv := FALSE;
   S_RTN1_STP2.SOL_Ret := FALSE;
   S_RTN1_STP2.M_Ready := FALSE;
   S_RTN1_STP2.T_CHK1 := T#0MS;
   S_RTN1_STP2.T_CHK2 := T#0MS;
   S_RTN1_STP2.PB_Lamp_CHK := FALSE;
   S_RTN1_STP2.PB_Error_Rst := FALSE;
   S_RTN1_STP2.M_FLICK := FALSE;
   S_RTN1_STP2.M_Adv_Err := FALSE;
   S_RTN1_STP2.M_Ret_Err := FALSE;
   S_RTN1_STP2.LP_Adv := FALSE;
   S_RTN1_STP2.LP_Ret := FALSE;
   S_RTN1_STP2.Visu_Adv := W#16#0;
   S_RTN1_STP2.Visu_Ret := W#16#0;
   S_RTN1_STP2.Error_T1.IN := FALSE;
   S_RTN1_STP2.Error_T1.PT := T#0MS;
   S_RTN1_STP2.Error_T1.Q := FALSE;
   S_RTN1_STP2.Error_T1.ET := T#0MS;
   S_RTN1_STP2.Error_T1.STATE := B#16#0;
   S_RTN1_STP2.Error_T1.STIME := T#0MS;
   S_RTN1_STP2.Error_T1.ATIME := T#0MS;
   S_RTN1_STP2.Error_T2.IN := FALSE;
   S_RTN1_STP2.Error_T2.PT := T#0MS;
   S_RTN1_STP2.Error_T2.Q := FALSE;
   S_RTN1_STP2.Error_T2.ET := T#0MS;
   S_RTN1_STP2.Error_T2.STATE := B#16#0;
   S_RTN1_STP2.Error_T2.STIME := T#0MS;
   S_RTN1_STP2.Error_T2.ATIME := T#0MS;
   S_RTN1_STP2.CHK_Aux1 := FALSE;
   S_RTN1_STP2.CHK_Aux2 := FALSE;
   S_RTN1_STP2.Error_T1_DN := FALSE;
   S_RTN1_STP2.Error_T2_DN := FALSE;
   S_RTN1_STP2.Adv_Memo := FALSE;
   S_RTN1_STP2.Visu_Adv_Arr[0] := FALSE;
   S_RTN1_STP2.Visu_Adv_Arr[1] := FALSE;
   S_RTN1_STP2.Visu_Adv_Arr[2] := FALSE;
   S_RTN1_STP2.Visu_Adv_Arr[3] := FALSE;
   S_RTN1_STP2.Visu_Adv_Arr[4] := FALSE;
   S_RTN1_STP2.Visu_Adv_Arr[5] := FALSE;
   S_RTN1_STP2.Visu_Adv_Arr[6] := FALSE;
   S_RTN1_STP2.Visu_Adv_Arr[7] := FALSE;
   S_RTN1_STP2.Visu_Adv_Arr[8] := FALSE;
   S_RTN1_STP2.Visu_Adv_Arr[9] := FALSE;
   S_RTN1_STP2.Visu_Adv_Arr[10] := FALSE;
   S_RTN1_STP2.Visu_Adv_Arr[11] := FALSE;
   S_RTN1_STP2.Visu_Adv_Arr[12] := FALSE;
   S_RTN1_STP2.Visu_Adv_Arr[13] := FALSE;
   S_RTN1_STP2.Visu_Adv_Arr[14] := FALSE;
   S_RTN1_STP2.Visu_Adv_Arr[15] := FALSE;
   S_RTN1_STP2.Visu_Ret_Arr[0] := FALSE;
   S_RTN1_STP2.Visu_Ret_Arr[1] := FALSE;
   S_RTN1_STP2.Visu_Ret_Arr[2] := FALSE;
   S_RTN1_STP2.Visu_Ret_Arr[3] := FALSE;
   S_RTN1_STP2.Visu_Ret_Arr[4] := FALSE;
   S_RTN1_STP2.Visu_Ret_Arr[5] := FALSE;
   S_RTN1_STP2.Visu_Ret_Arr[6] := FALSE;
   S_RTN1_STP2.Visu_Ret_Arr[7] := FALSE;
   S_RTN1_STP2.Visu_Ret_Arr[8] := FALSE;
   S_RTN1_STP2.Visu_Ret_Arr[9] := FALSE;
   S_RTN1_STP2.Visu_Ret_Arr[10] := FALSE;
   S_RTN1_STP2.Visu_Ret_Arr[11] := FALSE;
   S_RTN1_STP2.Visu_Ret_Arr[12] := FALSE;
   S_RTN1_STP2.Visu_Ret_Arr[13] := FALSE;
   S_RTN1_STP2.Visu_Ret_Arr[14] := FALSE;
   S_RTN1_STP2.Visu_Ret_Arr[15] := FALSE;
   S_RTN1_STP2.BLK_Move_Ret := 0;
   S_RTN1_STP2.Enable := FALSE;
   S_RTN1_STP2.Adv_End := FALSE;
   S_RTN1_STP2.Ret_End := FALSE;
   S_RTN1_STP3.Enable_Aux := FALSE;
   S_RTN1_STP3.Adv_Amount := 0;
   S_RTN1_STP3.Ret_Amount := 0;
   S_RTN1_STP3.LS_Adv1 := FALSE;
   S_RTN1_STP3.LS_Ret1 := FALSE;
   S_RTN1_STP3.LS_Adv2 := FALSE;
   S_RTN1_STP3.LS_Ret2 := FALSE;
   S_RTN1_STP3.LS_Adv3 := FALSE;
   S_RTN1_STP3.LS_Ret3 := FALSE;
   S_RTN1_STP3.LS_Adv4 := FALSE;
   S_RTN1_STP3.LS_Ret4 := FALSE;
   S_RTN1_STP3.SOL_Adv := FALSE;
   S_RTN1_STP3.SOL_Ret := FALSE;
   S_RTN1_STP3.M_Ready := FALSE;
   S_RTN1_STP3.T_CHK1 := T#0MS;
   S_RTN1_STP3.T_CHK2 := T#0MS;
   S_RTN1_STP3.PB_Lamp_CHK := FALSE;
   S_RTN1_STP3.PB_Error_Rst := FALSE;
   S_RTN1_STP3.M_FLICK := FALSE;
   S_RTN1_STP3.M_Adv_Err := FALSE;
   S_RTN1_STP3.M_Ret_Err := FALSE;
   S_RTN1_STP3.LP_Adv := FALSE;
   S_RTN1_STP3.LP_Ret := FALSE;
   S_RTN1_STP3.Visu_Adv := W#16#0;
   S_RTN1_STP3.Visu_Ret := W#16#0;
   S_RTN1_STP3.Error_T1.IN := FALSE;
   S_RTN1_STP3.Error_T1.PT := T#0MS;
   S_RTN1_STP3.Error_T1.Q := FALSE;
   S_RTN1_STP3.Error_T1.ET := T#0MS;
   S_RTN1_STP3.Error_T1.STATE := B#16#0;
   S_RTN1_STP3.Error_T1.STIME := T#0MS;
   S_RTN1_STP3.Error_T1.ATIME := T#0MS;
   S_RTN1_STP3.Error_T2.IN := FALSE;
   S_RTN1_STP3.Error_T2.PT := T#0MS;
   S_RTN1_STP3.Error_T2.Q := FALSE;
   S_RTN1_STP3.Error_T2.ET := T#0MS;
   S_RTN1_STP3.Error_T2.STATE := B#16#0;
   S_RTN1_STP3.Error_T2.STIME := T#0MS;
   S_RTN1_STP3.Error_T2.ATIME := T#0MS;
   S_RTN1_STP3.CHK_Aux1 := FALSE;
   S_RTN1_STP3.CHK_Aux2 := FALSE;
   S_RTN1_STP3.Error_T1_DN := FALSE;
   S_RTN1_STP3.Error_T2_DN := FALSE;
   S_RTN1_STP3.Adv_Memo := FALSE;
   S_RTN1_STP3.Visu_Adv_Arr[0] := FALSE;
   S_RTN1_STP3.Visu_Adv_Arr[1] := FALSE;
   S_RTN1_STP3.Visu_Adv_Arr[2] := FALSE;
   S_RTN1_STP3.Visu_Adv_Arr[3] := FALSE;
   S_RTN1_STP3.Visu_Adv_Arr[4] := FALSE;
   S_RTN1_STP3.Visu_Adv_Arr[5] := FALSE;
   S_RTN1_STP3.Visu_Adv_Arr[6] := FALSE;
   S_RTN1_STP3.Visu_Adv_Arr[7] := FALSE;
   S_RTN1_STP3.Visu_Adv_Arr[8] := FALSE;
   S_RTN1_STP3.Visu_Adv_Arr[9] := FALSE;
   S_RTN1_STP3.Visu_Adv_Arr[10] := FALSE;
   S_RTN1_STP3.Visu_Adv_Arr[11] := FALSE;
   S_RTN1_STP3.Visu_Adv_Arr[12] := FALSE;
   S_RTN1_STP3.Visu_Adv_Arr[13] := FALSE;
   S_RTN1_STP3.Visu_Adv_Arr[14] := FALSE;
   S_RTN1_STP3.Visu_Adv_Arr[15] := FALSE;
   S_RTN1_STP3.Visu_Ret_Arr[0] := FALSE;
   S_RTN1_STP3.Visu_Ret_Arr[1] := FALSE;
   S_RTN1_STP3.Visu_Ret_Arr[2] := FALSE;
   S_RTN1_STP3.Visu_Ret_Arr[3] := FALSE;
   S_RTN1_STP3.Visu_Ret_Arr[4] := FALSE;
   S_RTN1_STP3.Visu_Ret_Arr[5] := FALSE;
   S_RTN1_STP3.Visu_Ret_Arr[6] := FALSE;
   S_RTN1_STP3.Visu_Ret_Arr[7] := FALSE;
   S_RTN1_STP3.Visu_Ret_Arr[8] := FALSE;
   S_RTN1_STP3.Visu_Ret_Arr[9] := FALSE;
   S_RTN1_STP3.Visu_Ret_Arr[10] := FALSE;
   S_RTN1_STP3.Visu_Ret_Arr[11] := FALSE;
   S_RTN1_STP3.Visu_Ret_Arr[12] := FALSE;
   S_RTN1_STP3.Visu_Ret_Arr[13] := FALSE;
   S_RTN1_STP3.Visu_Ret_Arr[14] := FALSE;
   S_RTN1_STP3.Visu_Ret_Arr[15] := FALSE;
   S_RTN1_STP3.BLK_Move_Ret := 0;
   S_RTN1_STP3.Enable := FALSE;
   S_RTN1_STP3.Adv_End := FALSE;
   S_RTN1_STP3.Ret_End := FALSE;
   S_RTN1_STP4.Enable_Aux := FALSE;
   S_RTN1_STP4.Adv_Amount := 0;
   S_RTN1_STP4.Ret_Amount := 0;
   S_RTN1_STP4.LS_Adv1 := FALSE;
   S_RTN1_STP4.LS_Ret1 := FALSE;
   S_RTN1_STP4.LS_Adv2 := FALSE;
   S_RTN1_STP4.LS_Ret2 := FALSE;
   S_RTN1_STP4.LS_Adv3 := FALSE;
   S_RTN1_STP4.LS_Ret3 := FALSE;
   S_RTN1_STP4.LS_Adv4 := FALSE;
   S_RTN1_STP4.LS_Ret4 := FALSE;
   S_RTN1_STP4.SOL_Adv := FALSE;
   S_RTN1_STP4.SOL_Ret := FALSE;
   S_RTN1_STP4.M_Ready := FALSE;
   S_RTN1_STP4.T_CHK1 := T#0MS;
   S_RTN1_STP4.T_CHK2 := T#0MS;
   S_RTN1_STP4.PB_Lamp_CHK := FALSE;
   S_RTN1_STP4.PB_Error_Rst := FALSE;
   S_RTN1_STP4.M_FLICK := FALSE;
   S_RTN1_STP4.M_Adv_Err := FALSE;
   S_RTN1_STP4.M_Ret_Err := FALSE;
   S_RTN1_STP4.LP_Adv := FALSE;
   S_RTN1_STP4.LP_Ret := FALSE;
   S_RTN1_STP4.Visu_Adv := W#16#0;
   S_RTN1_STP4.Visu_Ret := W#16#0;
   S_RTN1_STP4.Error_T1.IN := FALSE;
   S_RTN1_STP4.Error_T1.PT := T#0MS;
   S_RTN1_STP4.Error_T1.Q := FALSE;
   S_RTN1_STP4.Error_T1.ET := T#0MS;
   S_RTN1_STP4.Error_T1.STATE := B#16#0;
   S_RTN1_STP4.Error_T1.STIME := T#0MS;
   S_RTN1_STP4.Error_T1.ATIME := T#0MS;
   S_RTN1_STP4.Error_T2.IN := FALSE;
   S_RTN1_STP4.Error_T2.PT := T#0MS;
   S_RTN1_STP4.Error_T2.Q := FALSE;
   S_RTN1_STP4.Error_T2.ET := T#0MS;
   S_RTN1_STP4.Error_T2.STATE := B#16#0;
   S_RTN1_STP4.Error_T2.STIME := T#0MS;
   S_RTN1_STP4.Error_T2.ATIME := T#0MS;
   S_RTN1_STP4.CHK_Aux1 := FALSE;
   S_RTN1_STP4.CHK_Aux2 := FALSE;
   S_RTN1_STP4.Error_T1_DN := FALSE;
   S_RTN1_STP4.Error_T2_DN := FALSE;
   S_RTN1_STP4.Adv_Memo := FALSE;
   S_RTN1_STP4.Visu_Adv_Arr[0] := FALSE;
   S_RTN1_STP4.Visu_Adv_Arr[1] := FALSE;
   S_RTN1_STP4.Visu_Adv_Arr[2] := FALSE;
   S_RTN1_STP4.Visu_Adv_Arr[3] := FALSE;
   S_RTN1_STP4.Visu_Adv_Arr[4] := FALSE;
   S_RTN1_STP4.Visu_Adv_Arr[5] := FALSE;
   S_RTN1_STP4.Visu_Adv_Arr[6] := FALSE;
   S_RTN1_STP4.Visu_Adv_Arr[7] := FALSE;
   S_RTN1_STP4.Visu_Adv_Arr[8] := FALSE;
   S_RTN1_STP4.Visu_Adv_Arr[9] := FALSE;
   S_RTN1_STP4.Visu_Adv_Arr[10] := FALSE;
   S_RTN1_STP4.Visu_Adv_Arr[11] := FALSE;
   S_RTN1_STP4.Visu_Adv_Arr[12] := FALSE;
   S_RTN1_STP4.Visu_Adv_Arr[13] := FALSE;
   S_RTN1_STP4.Visu_Adv_Arr[14] := FALSE;
   S_RTN1_STP4.Visu_Adv_Arr[15] := FALSE;
   S_RTN1_STP4.Visu_Ret_Arr[0] := FALSE;
   S_RTN1_STP4.Visu_Ret_Arr[1] := FALSE;
   S_RTN1_STP4.Visu_Ret_Arr[2] := FALSE;
   S_RTN1_STP4.Visu_Ret_Arr[3] := FALSE;
   S_RTN1_STP4.Visu_Ret_Arr[4] := FALSE;
   S_RTN1_STP4.Visu_Ret_Arr[5] := FALSE;
   S_RTN1_STP4.Visu_Ret_Arr[6] := FALSE;
   S_RTN1_STP4.Visu_Ret_Arr[7] := FALSE;
   S_RTN1_STP4.Visu_Ret_Arr[8] := FALSE;
   S_RTN1_STP4.Visu_Ret_Arr[9] := FALSE;
   S_RTN1_STP4.Visu_Ret_Arr[10] := FALSE;
   S_RTN1_STP4.Visu_Ret_Arr[11] := FALSE;
   S_RTN1_STP4.Visu_Ret_Arr[12] := FALSE;
   S_RTN1_STP4.Visu_Ret_Arr[13] := FALSE;
   S_RTN1_STP4.Visu_Ret_Arr[14] := FALSE;
   S_RTN1_STP4.Visu_Ret_Arr[15] := FALSE;
   S_RTN1_STP4.BLK_Move_Ret := 0;
   S_RTN1_STP4.Enable := FALSE;
   S_RTN1_STP4.Adv_End := FALSE;
   S_RTN1_STP4.Ret_End := FALSE;
   S_RTN2_STP1.Enable_Aux := FALSE;
   S_RTN2_STP1.Adv_Amount := 0;
   S_RTN2_STP1.Ret_Amount := 0;
   S_RTN2_STP1.LS_Adv1 := FALSE;
   S_RTN2_STP1.LS_Ret1 := FALSE;
   S_RTN2_STP1.LS_Adv2 := FALSE;
   S_RTN2_STP1.LS_Ret2 := FALSE;
   S_RTN2_STP1.LS_Adv3 := FALSE;
   S_RTN2_STP1.LS_Ret3 := FALSE;
   S_RTN2_STP1.LS_Adv4 := FALSE;
   S_RTN2_STP1.LS_Ret4 := FALSE;
   S_RTN2_STP1.SOL_Adv := FALSE;
   S_RTN2_STP1.SOL_Ret := FALSE;
   S_RTN2_STP1.M_Ready := FALSE;
   S_RTN2_STP1.T_CHK1 := T#0MS;
   S_RTN2_STP1.T_CHK2 := T#0MS;
   S_RTN2_STP1.PB_Lamp_CHK := FALSE;
   S_RTN2_STP1.PB_Error_Rst := FALSE;
   S_RTN2_STP1.M_FLICK := FALSE;
   S_RTN2_STP1.M_Adv_Err := FALSE;
   S_RTN2_STP1.M_Ret_Err := FALSE;
   S_RTN2_STP1.LP_Adv := FALSE;
   S_RTN2_STP1.LP_Ret := FALSE;
   S_RTN2_STP1.Visu_Adv := W#16#0;
   S_RTN2_STP1.Visu_Ret := W#16#0;
   S_RTN2_STP1.Error_T1.IN := FALSE;
   S_RTN2_STP1.Error_T1.PT := T#0MS;
   S_RTN2_STP1.Error_T1.Q := FALSE;
   S_RTN2_STP1.Error_T1.ET := T#0MS;
   S_RTN2_STP1.Error_T1.STATE := B#16#0;
   S_RTN2_STP1.Error_T1.STIME := T#0MS;
   S_RTN2_STP1.Error_T1.ATIME := T#0MS;
   S_RTN2_STP1.Error_T2.IN := FALSE;
   S_RTN2_STP1.Error_T2.PT := T#0MS;
   S_RTN2_STP1.Error_T2.Q := FALSE;
   S_RTN2_STP1.Error_T2.ET := T#0MS;
   S_RTN2_STP1.Error_T2.STATE := B#16#0;
   S_RTN2_STP1.Error_T2.STIME := T#0MS;
   S_RTN2_STP1.Error_T2.ATIME := T#0MS;
   S_RTN2_STP1.CHK_Aux1 := FALSE;
   S_RTN2_STP1.CHK_Aux2 := FALSE;
   S_RTN2_STP1.Error_T1_DN := FALSE;
   S_RTN2_STP1.Error_T2_DN := FALSE;
   S_RTN2_STP1.Adv_Memo := FALSE;
   S_RTN2_STP1.Visu_Adv_Arr[0] := FALSE;
   S_RTN2_STP1.Visu_Adv_Arr[1] := FALSE;
   S_RTN2_STP1.Visu_Adv_Arr[2] := FALSE;
   S_RTN2_STP1.Visu_Adv_Arr[3] := FALSE;
   S_RTN2_STP1.Visu_Adv_Arr[4] := FALSE;
   S_RTN2_STP1.Visu_Adv_Arr[5] := FALSE;
   S_RTN2_STP1.Visu_Adv_Arr[6] := FALSE;
   S_RTN2_STP1.Visu_Adv_Arr[7] := FALSE;
   S_RTN2_STP1.Visu_Adv_Arr[8] := FALSE;
   S_RTN2_STP1.Visu_Adv_Arr[9] := FALSE;
   S_RTN2_STP1.Visu_Adv_Arr[10] := FALSE;
   S_RTN2_STP1.Visu_Adv_Arr[11] := FALSE;
   S_RTN2_STP1.Visu_Adv_Arr[12] := FALSE;
   S_RTN2_STP1.Visu_Adv_Arr[13] := FALSE;
   S_RTN2_STP1.Visu_Adv_Arr[14] := FALSE;
   S_RTN2_STP1.Visu_Adv_Arr[15] := FALSE;
   S_RTN2_STP1.Visu_Ret_Arr[0] := FALSE;
   S_RTN2_STP1.Visu_Ret_Arr[1] := FALSE;
   S_RTN2_STP1.Visu_Ret_Arr[2] := FALSE;
   S_RTN2_STP1.Visu_Ret_Arr[3] := FALSE;
   S_RTN2_STP1.Visu_Ret_Arr[4] := FALSE;
   S_RTN2_STP1.Visu_Ret_Arr[5] := FALSE;
   S_RTN2_STP1.Visu_Ret_Arr[6] := FALSE;
   S_RTN2_STP1.Visu_Ret_Arr[7] := FALSE;
   S_RTN2_STP1.Visu_Ret_Arr[8] := FALSE;
   S_RTN2_STP1.Visu_Ret_Arr[9] := FALSE;
   S_RTN2_STP1.Visu_Ret_Arr[10] := FALSE;
   S_RTN2_STP1.Visu_Ret_Arr[11] := FALSE;
   S_RTN2_STP1.Visu_Ret_Arr[12] := FALSE;
   S_RTN2_STP1.Visu_Ret_Arr[13] := FALSE;
   S_RTN2_STP1.Visu_Ret_Arr[14] := FALSE;
   S_RTN2_STP1.Visu_Ret_Arr[15] := FALSE;
   S_RTN2_STP1.BLK_Move_Ret := 0;
   S_RTN2_STP1.Enable := FALSE;
   S_RTN2_STP1.Adv_End := FALSE;
   S_RTN2_STP1.Ret_End := FALSE;
   S_RTN2_STP2.Enable_Aux := FALSE;
   S_RTN2_STP2.Adv_Amount := 0;
   S_RTN2_STP2.Ret_Amount := 0;
   S_RTN2_STP2.LS_Adv1 := FALSE;
   S_RTN2_STP2.LS_Ret1 := FALSE;
   S_RTN2_STP2.LS_Adv2 := FALSE;
   S_RTN2_STP2.LS_Ret2 := FALSE;
   S_RTN2_STP2.LS_Adv3 := FALSE;
   S_RTN2_STP2.LS_Ret3 := FALSE;
   S_RTN2_STP2.LS_Adv4 := FALSE;
   S_RTN2_STP2.LS_Ret4 := FALSE;
   S_RTN2_STP2.SOL_Adv := FALSE;
   S_RTN2_STP2.SOL_Ret := FALSE;
   S_RTN2_STP2.M_Ready := FALSE;
   S_RTN2_STP2.T_CHK1 := T#0MS;
   S_RTN2_STP2.T_CHK2 := T#0MS;
   S_RTN2_STP2.PB_Lamp_CHK := FALSE;
   S_RTN2_STP2.PB_Error_Rst := FALSE;
   S_RTN2_STP2.M_FLICK := FALSE;
   S_RTN2_STP2.M_Adv_Err := FALSE;
   S_RTN2_STP2.M_Ret_Err := FALSE;
   S_RTN2_STP2.LP_Adv := FALSE;
   S_RTN2_STP2.LP_Ret := FALSE;
   S_RTN2_STP2.Visu_Adv := W#16#0;
   S_RTN2_STP2.Visu_Ret := W#16#0;
   S_RTN2_STP2.Error_T1.IN := FALSE;
   S_RTN2_STP2.Error_T1.PT := T#0MS;
   S_RTN2_STP2.Error_T1.Q := FALSE;
   S_RTN2_STP2.Error_T1.ET := T#0MS;
   S_RTN2_STP2.Error_T1.STATE := B#16#0;
   S_RTN2_STP2.Error_T1.STIME := T#0MS;
   S_RTN2_STP2.Error_T1.ATIME := T#0MS;
   S_RTN2_STP2.Error_T2.IN := FALSE;
   S_RTN2_STP2.Error_T2.PT := T#0MS;
   S_RTN2_STP2.Error_T2.Q := FALSE;
   S_RTN2_STP2.Error_T2.ET := T#0MS;
   S_RTN2_STP2.Error_T2.STATE := B#16#0;
   S_RTN2_STP2.Error_T2.STIME := T#0MS;
   S_RTN2_STP2.Error_T2.ATIME := T#0MS;
   S_RTN2_STP2.CHK_Aux1 := FALSE;
   S_RTN2_STP2.CHK_Aux2 := FALSE;
   S_RTN2_STP2.Error_T1_DN := FALSE;
   S_RTN2_STP2.Error_T2_DN := FALSE;
   S_RTN2_STP2.Adv_Memo := FALSE;
   S_RTN2_STP2.Visu_Adv_Arr[0] := FALSE;
   S_RTN2_STP2.Visu_Adv_Arr[1] := FALSE;
   S_RTN2_STP2.Visu_Adv_Arr[2] := FALSE;
   S_RTN2_STP2.Visu_Adv_Arr[3] := FALSE;
   S_RTN2_STP2.Visu_Adv_Arr[4] := FALSE;
   S_RTN2_STP2.Visu_Adv_Arr[5] := FALSE;
   S_RTN2_STP2.Visu_Adv_Arr[6] := FALSE;
   S_RTN2_STP2.Visu_Adv_Arr[7] := FALSE;
   S_RTN2_STP2.Visu_Adv_Arr[8] := FALSE;
   S_RTN2_STP2.Visu_Adv_Arr[9] := FALSE;
   S_RTN2_STP2.Visu_Adv_Arr[10] := FALSE;
   S_RTN2_STP2.Visu_Adv_Arr[11] := FALSE;
   S_RTN2_STP2.Visu_Adv_Arr[12] := FALSE;
   S_RTN2_STP2.Visu_Adv_Arr[13] := FALSE;
   S_RTN2_STP2.Visu_Adv_Arr[14] := FALSE;
   S_RTN2_STP2.Visu_Adv_Arr[15] := FALSE;
   S_RTN2_STP2.Visu_Ret_Arr[0] := FALSE;
   S_RTN2_STP2.Visu_Ret_Arr[1] := FALSE;
   S_RTN2_STP2.Visu_Ret_Arr[2] := FALSE;
   S_RTN2_STP2.Visu_Ret_Arr[3] := FALSE;
   S_RTN2_STP2.Visu_Ret_Arr[4] := FALSE;
   S_RTN2_STP2.Visu_Ret_Arr[5] := FALSE;
   S_RTN2_STP2.Visu_Ret_Arr[6] := FALSE;
   S_RTN2_STP2.Visu_Ret_Arr[7] := FALSE;
   S_RTN2_STP2.Visu_Ret_Arr[8] := FALSE;
   S_RTN2_STP2.Visu_Ret_Arr[9] := FALSE;
   S_RTN2_STP2.Visu_Ret_Arr[10] := FALSE;
   S_RTN2_STP2.Visu_Ret_Arr[11] := FALSE;
   S_RTN2_STP2.Visu_Ret_Arr[12] := FALSE;
   S_RTN2_STP2.Visu_Ret_Arr[13] := FALSE;
   S_RTN2_STP2.Visu_Ret_Arr[14] := FALSE;
   S_RTN2_STP2.Visu_Ret_Arr[15] := FALSE;
   S_RTN2_STP2.BLK_Move_Ret := 0;
   S_RTN2_STP2.Enable := FALSE;
   S_RTN2_STP2.Adv_End := FALSE;
   S_RTN2_STP2.Ret_End := FALSE;
   S_RTN3_STP1.Enable_Aux := FALSE;
   S_RTN3_STP1.Adv_Amount := 0;
   S_RTN3_STP1.Ret_Amount := 0;
   S_RTN3_STP1.LS_Adv1 := FALSE;
   S_RTN3_STP1.LS_Ret1 := FALSE;
   S_RTN3_STP1.LS_Adv2 := FALSE;
   S_RTN3_STP1.LS_Ret2 := FALSE;
   S_RTN3_STP1.LS_Adv3 := FALSE;
   S_RTN3_STP1.LS_Ret3 := FALSE;
   S_RTN3_STP1.LS_Adv4 := FALSE;
   S_RTN3_STP1.LS_Ret4 := FALSE;
   S_RTN3_STP1.SOL_Adv := FALSE;
   S_RTN3_STP1.SOL_Ret := FALSE;
   S_RTN3_STP1.M_Ready := FALSE;
   S_RTN3_STP1.T_CHK1 := T#0MS;
   S_RTN3_STP1.T_CHK2 := T#0MS;
   S_RTN3_STP1.PB_Lamp_CHK := FALSE;
   S_RTN3_STP1.PB_Error_Rst := FALSE;
   S_RTN3_STP1.M_FLICK := FALSE;
   S_RTN3_STP1.M_Adv_Err := FALSE;
   S_RTN3_STP1.M_Ret_Err := FALSE;
   S_RTN3_STP1.LP_Adv := FALSE;
   S_RTN3_STP1.LP_Ret := FALSE;
   S_RTN3_STP1.Visu_Adv := W#16#0;
   S_RTN3_STP1.Visu_Ret := W#16#0;
   S_RTN3_STP1.Error_T1.IN := FALSE;
   S_RTN3_STP1.Error_T1.PT := T#0MS;
   S_RTN3_STP1.Error_T1.Q := FALSE;
   S_RTN3_STP1.Error_T1.ET := T#0MS;
   S_RTN3_STP1.Error_T1.STATE := B#16#0;
   S_RTN3_STP1.Error_T1.STIME := T#0MS;
   S_RTN3_STP1.Error_T1.ATIME := T#0MS;
   S_RTN3_STP1.Error_T2.IN := FALSE;
   S_RTN3_STP1.Error_T2.PT := T#0MS;
   S_RTN3_STP1.Error_T2.Q := FALSE;
   S_RTN3_STP1.Error_T2.ET := T#0MS;
   S_RTN3_STP1.Error_T2.STATE := B#16#0;
   S_RTN3_STP1.Error_T2.STIME := T#0MS;
   S_RTN3_STP1.Error_T2.ATIME := T#0MS;
   S_RTN3_STP1.CHK_Aux1 := FALSE;
   S_RTN3_STP1.CHK_Aux2 := FALSE;
   S_RTN3_STP1.Error_T1_DN := FALSE;
   S_RTN3_STP1.Error_T2_DN := FALSE;
   S_RTN3_STP1.Adv_Memo := FALSE;
   S_RTN3_STP1.Visu_Adv_Arr[0] := FALSE;
   S_RTN3_STP1.Visu_Adv_Arr[1] := FALSE;
   S_RTN3_STP1.Visu_Adv_Arr[2] := FALSE;
   S_RTN3_STP1.Visu_Adv_Arr[3] := FALSE;
   S_RTN3_STP1.Visu_Adv_Arr[4] := FALSE;
   S_RTN3_STP1.Visu_Adv_Arr[5] := FALSE;
   S_RTN3_STP1.Visu_Adv_Arr[6] := FALSE;
   S_RTN3_STP1.Visu_Adv_Arr[7] := FALSE;
   S_RTN3_STP1.Visu_Adv_Arr[8] := FALSE;
   S_RTN3_STP1.Visu_Adv_Arr[9] := FALSE;
   S_RTN3_STP1.Visu_Adv_Arr[10] := FALSE;
   S_RTN3_STP1.Visu_Adv_Arr[11] := FALSE;
   S_RTN3_STP1.Visu_Adv_Arr[12] := FALSE;
   S_RTN3_STP1.Visu_Adv_Arr[13] := FALSE;
   S_RTN3_STP1.Visu_Adv_Arr[14] := FALSE;
   S_RTN3_STP1.Visu_Adv_Arr[15] := FALSE;
   S_RTN3_STP1.Visu_Ret_Arr[0] := FALSE;
   S_RTN3_STP1.Visu_Ret_Arr[1] := FALSE;
   S_RTN3_STP1.Visu_Ret_Arr[2] := FALSE;
   S_RTN3_STP1.Visu_Ret_Arr[3] := FALSE;
   S_RTN3_STP1.Visu_Ret_Arr[4] := FALSE;
   S_RTN3_STP1.Visu_Ret_Arr[5] := FALSE;
   S_RTN3_STP1.Visu_Ret_Arr[6] := FALSE;
   S_RTN3_STP1.Visu_Ret_Arr[7] := FALSE;
   S_RTN3_STP1.Visu_Ret_Arr[8] := FALSE;
   S_RTN3_STP1.Visu_Ret_Arr[9] := FALSE;
   S_RTN3_STP1.Visu_Ret_Arr[10] := FALSE;
   S_RTN3_STP1.Visu_Ret_Arr[11] := FALSE;
   S_RTN3_STP1.Visu_Ret_Arr[12] := FALSE;
   S_RTN3_STP1.Visu_Ret_Arr[13] := FALSE;
   S_RTN3_STP1.Visu_Ret_Arr[14] := FALSE;
   S_RTN3_STP1.Visu_Ret_Arr[15] := FALSE;
   S_RTN3_STP1.BLK_Move_Ret := 0;
   S_RTN3_STP1.Enable := FALSE;
   S_RTN3_STP1.Adv_End := FALSE;
   S_RTN3_STP1.Ret_End := FALSE;
   S_RTN3_STP2.Enable_Aux := FALSE;
   S_RTN3_STP2.Adv_Amount := 0;
   S_RTN3_STP2.Ret_Amount := 0;
   S_RTN3_STP2.LS_Adv1 := FALSE;
   S_RTN3_STP2.LS_Ret1 := FALSE;
   S_RTN3_STP2.LS_Adv2 := FALSE;
   S_RTN3_STP2.LS_Ret2 := FALSE;
   S_RTN3_STP2.LS_Adv3 := FALSE;
   S_RTN3_STP2.LS_Ret3 := FALSE;
   S_RTN3_STP2.LS_Adv4 := FALSE;
   S_RTN3_STP2.LS_Ret4 := FALSE;
   S_RTN3_STP2.SOL_Adv := FALSE;
   S_RTN3_STP2.SOL_Ret := FALSE;
   S_RTN3_STP2.M_Ready := FALSE;
   S_RTN3_STP2.T_CHK1 := T#0MS;
   S_RTN3_STP2.T_CHK2 := T#0MS;
   S_RTN3_STP2.PB_Lamp_CHK := FALSE;
   S_RTN3_STP2.PB_Error_Rst := FALSE;
   S_RTN3_STP2.M_FLICK := FALSE;
   S_RTN3_STP2.M_Adv_Err := FALSE;
   S_RTN3_STP2.M_Ret_Err := FALSE;
   S_RTN3_STP2.LP_Adv := FALSE;
   S_RTN3_STP2.LP_Ret := FALSE;
   S_RTN3_STP2.Visu_Adv := W#16#0;
   S_RTN3_STP2.Visu_Ret := W#16#0;
   S_RTN3_STP2.Error_T1.IN := FALSE;
   S_RTN3_STP2.Error_T1.PT := T#0MS;
   S_RTN3_STP2.Error_T1.Q := FALSE;
   S_RTN3_STP2.Error_T1.ET := T#0MS;
   S_RTN3_STP2.Error_T1.STATE := B#16#0;
   S_RTN3_STP2.Error_T1.STIME := T#0MS;
   S_RTN3_STP2.Error_T1.ATIME := T#0MS;
   S_RTN3_STP2.Error_T2.IN := FALSE;
   S_RTN3_STP2.Error_T2.PT := T#0MS;
   S_RTN3_STP2.Error_T2.Q := FALSE;
   S_RTN3_STP2.Error_T2.ET := T#0MS;
   S_RTN3_STP2.Error_T2.STATE := B#16#0;
   S_RTN3_STP2.Error_T2.STIME := T#0MS;
   S_RTN3_STP2.Error_T2.ATIME := T#0MS;
   S_RTN3_STP2.CHK_Aux1 := FALSE;
   S_RTN3_STP2.CHK_Aux2 := FALSE;
   S_RTN3_STP2.Error_T1_DN := FALSE;
   S_RTN3_STP2.Error_T2_DN := FALSE;
   S_RTN3_STP2.Adv_Memo := FALSE;
   S_RTN3_STP2.Visu_Adv_Arr[0] := FALSE;
   S_RTN3_STP2.Visu_Adv_Arr[1] := FALSE;
   S_RTN3_STP2.Visu_Adv_Arr[2] := FALSE;
   S_RTN3_STP2.Visu_Adv_Arr[3] := FALSE;
   S_RTN3_STP2.Visu_Adv_Arr[4] := FALSE;
   S_RTN3_STP2.Visu_Adv_Arr[5] := FALSE;
   S_RTN3_STP2.Visu_Adv_Arr[6] := FALSE;
   S_RTN3_STP2.Visu_Adv_Arr[7] := FALSE;
   S_RTN3_STP2.Visu_Adv_Arr[8] := FALSE;
   S_RTN3_STP2.Visu_Adv_Arr[9] := FALSE;
   S_RTN3_STP2.Visu_Adv_Arr[10] := FALSE;
   S_RTN3_STP2.Visu_Adv_Arr[11] := FALSE;
   S_RTN3_STP2.Visu_Adv_Arr[12] := FALSE;
   S_RTN3_STP2.Visu_Adv_Arr[13] := FALSE;
   S_RTN3_STP2.Visu_Adv_Arr[14] := FALSE;
   S_RTN3_STP2.Visu_Adv_Arr[15] := FALSE;
   S_RTN3_STP2.Visu_Ret_Arr[0] := FALSE;
   S_RTN3_STP2.Visu_Ret_Arr[1] := FALSE;
   S_RTN3_STP2.Visu_Ret_Arr[2] := FALSE;
   S_RTN3_STP2.Visu_Ret_Arr[3] := FALSE;
   S_RTN3_STP2.Visu_Ret_Arr[4] := FALSE;
   S_RTN3_STP2.Visu_Ret_Arr[5] := FALSE;
   S_RTN3_STP2.Visu_Ret_Arr[6] := FALSE;
   S_RTN3_STP2.Visu_Ret_Arr[7] := FALSE;
   S_RTN3_STP2.Visu_Ret_Arr[8] := FALSE;
   S_RTN3_STP2.Visu_Ret_Arr[9] := FALSE;
   S_RTN3_STP2.Visu_Ret_Arr[10] := FALSE;
   S_RTN3_STP2.Visu_Ret_Arr[11] := FALSE;
   S_RTN3_STP2.Visu_Ret_Arr[12] := FALSE;
   S_RTN3_STP2.Visu_Ret_Arr[13] := FALSE;
   S_RTN3_STP2.Visu_Ret_Arr[14] := FALSE;
   S_RTN3_STP2.Visu_Ret_Arr[15] := FALSE;
   S_RTN3_STP2.BLK_Move_Ret := 0;
   S_RTN3_STP2.Enable := FALSE;
   S_RTN3_STP2.Adv_End := FALSE;
   S_RTN3_STP2.Ret_End := FALSE;
END_DATA_BLOCK

FUNCTION FC 121 : VOID
TITLE =
VERSION : 0.1

BEGIN
NETWORK
TITLE =

END_FUNCTION

FUNCTION_BLOCK FB 122
TITLE =
VERSION : 0.1

BEGIN
NETWORK
TITLE =리턴1 이상

NETWORK
TITLE =
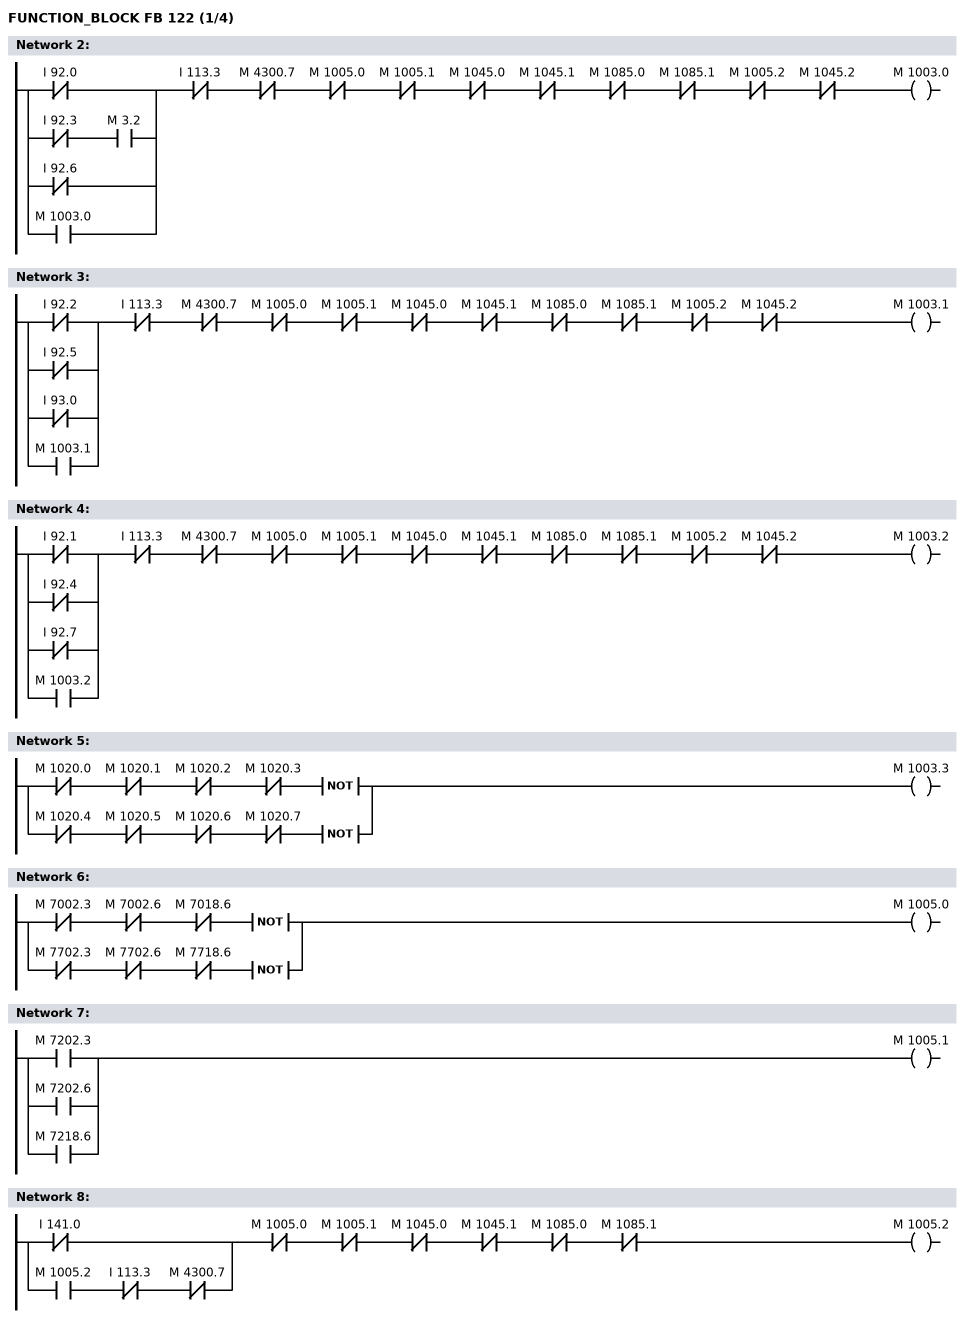

      A(    ;
      ON    I     92.0;
      O     ;
      AN    I     92.3;
      A     M      3.2;
      ON    I     92.6;
      O     M   1003.0;
      )     ;
      AN    I    113.3;
      AN    M   4300.7;
      AN    M   1005.0;
      AN    M   1005.1;
      AN    M   1045.0;
      AN    M   1045.1;
      AN    M   1085.0;
      AN    M   1085.1;
      AN    M   1005.2;
      AN    M   1045.2;
      =     M   1003.0;
NETWORK
TITLE =

      A(    ;
      ON    I     92.2;
      ON    I     92.5;
      ON    I     93.0;
      O     M   1003.1;
      )     ;
      AN    I    113.3;
      AN    M   4300.7;
      AN    M   1005.0;
      AN    M   1005.1;
      AN    M   1045.0;
      AN    M   1045.1;
      AN    M   1085.0;
      AN    M   1085.1;
      AN    M   1005.2;
      AN    M   1045.2;
      =     M   1003.1;
NETWORK
TITLE =

      A(    ;
      ON    I     92.1;
      ON    I     92.4;
      ON    I     92.7;
      O     M   1003.2;
      )     ;
      AN    I    113.3;
      AN    M   4300.7;
      AN    M   1005.0;
      AN    M   1005.1;
      AN    M   1045.0;
      AN    M   1045.1;
      AN    M   1085.0;
      AN    M   1085.1;
      AN    M   1005.2;
      AN    M   1045.2;
      =     M   1003.2;
NETWORK
TITLE =

      AN    M   1020.0;
      AN    M   1020.1;
      AN    M   1020.2;
      AN    M   1020.3;
      NOT   ;
      O(    ;
      AN    M   1020.4;
      AN    M   1020.5;
      AN    M   1020.6;
      AN    M   1020.7;
      NOT   ;
      )     ;
      =     M   1003.3;
NETWORK
TITLE =

      AN    M   7002.3;
      AN    M   7002.6;
      AN    M   7018.6;
      NOT   ;
      O(    ;
      AN    M   7702.3;
      AN    M   7702.6;
      AN    M   7718.6;
      NOT   ;
      )     ;
      =     M   1005.0;
NETWORK
TITLE =

      O     M   7202.3;
      O     M   7202.6;
      O     M   7218.6;
      =     M   1005.1;
NETWORK
TITLE =

      A(    ;
      ON    I    141.0;
      O     ;
      A     M   1005.2;
      AN    I    113.3;
      AN    M   4300.7;
      )     ;
      AN    M   1005.0;
      AN    M   1005.1;
      AN    M   1045.0;
      AN    M   1045.1;
      AN    M   1085.0;
      AN    M   1085.1;
      =     M   1005.2;
NETWORK
TITLE =
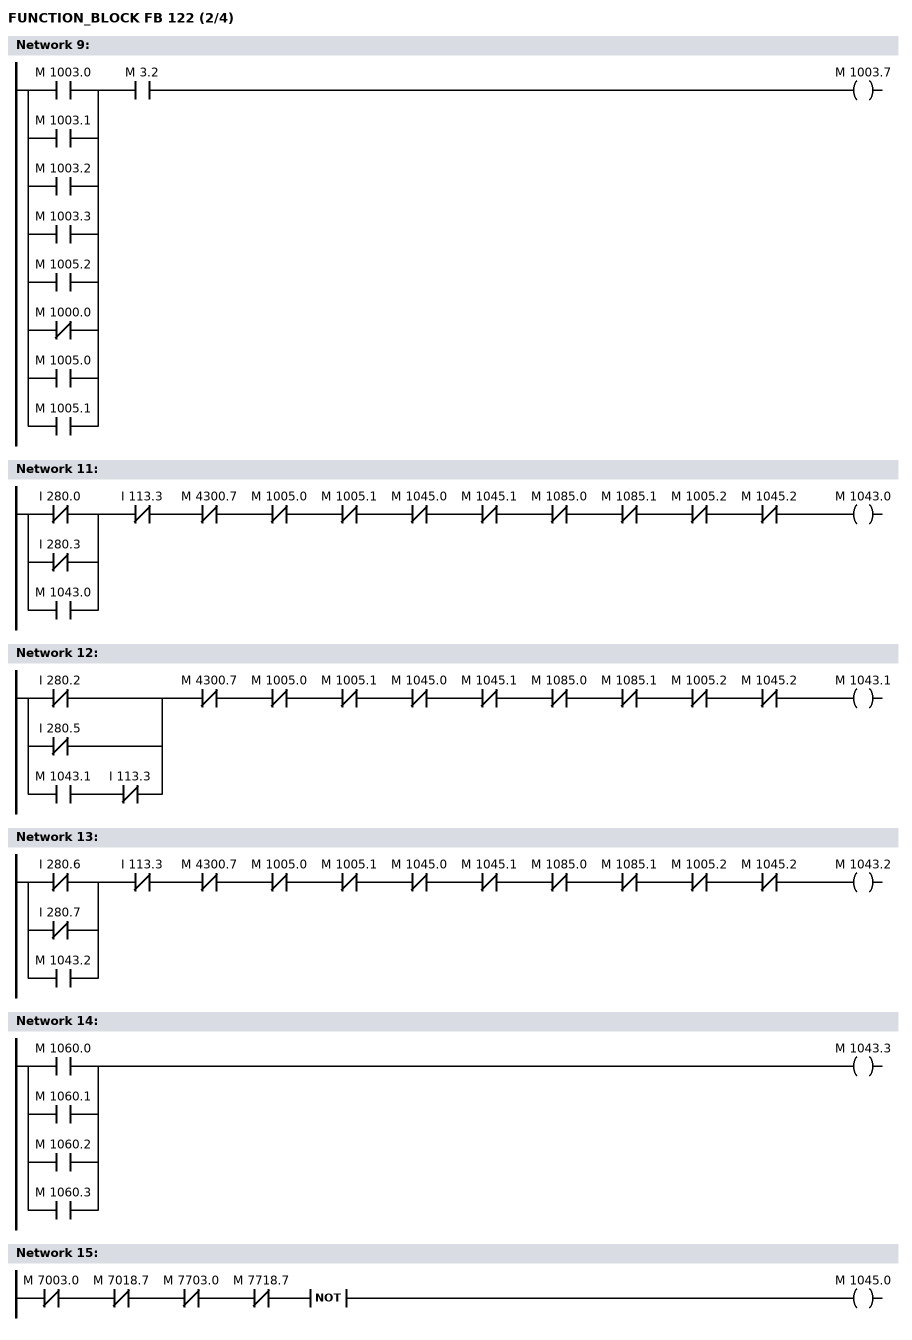

      A(    ;
      O     M   1003.0;
      O     M   1003.1;
      O     M   1003.2;
      O     M   1003.3;
      O     M   1005.2;
      ON    M   1000.0;
      O     M   1005.0;
      O     M   1005.1;
      )     ;
      A     M      3.2;
      =     M   1003.7;
NETWORK
TITLE =리턴2 이상

NETWORK
TITLE =

      A(    ;
      ON    I    280.0;
      ON    I    280.3;
      O     M   1043.0;
      )     ;
      AN    I    113.3;
      AN    M   4300.7;
      AN    M   1005.0;
      AN    M   1005.1;
      AN    M   1045.0;
      AN    M   1045.1;
      AN    M   1085.0;
      AN    M   1085.1;
      AN    M   1005.2;
      AN    M   1045.2;
      =     M   1043.0;
NETWORK
TITLE =

      A(    ;
      ON    I    280.2;
      ON    I    280.5;
      O     ;
      A     M   1043.1;
      AN    I    113.3;
      )     ;
      AN    M   4300.7;
      AN    M   1005.0;
      AN    M   1005.1;
      AN    M   1045.0;
      AN    M   1045.1;
      AN    M   1085.0;
      AN    M   1085.1;
      AN    M   1005.2;
      AN    M   1045.2;
      =     M   1043.1;
NETWORK
TITLE =

      A(    ;
      ON    I    280.6;
      ON    I    280.7;
      O     M   1043.2;
      )     ;
      AN    I    113.3;
      AN    M   4300.7;
      AN    M   1005.0;
      AN    M   1005.1;
      AN    M   1045.0;
      AN    M   1045.1;
      AN    M   1085.0;
      AN    M   1085.1;
      AN    M   1005.2;
      AN    M   1045.2;
      =     M   1043.2;
NETWORK
TITLE =

      O     M   1060.0;
      O     M   1060.1;
      O     M   1060.2;
      O     M   1060.3;
      =     M   1043.3;
NETWORK
TITLE =

      AN    M   7003.0;
      AN    M   7018.7;
      AN    M   7703.0;
      AN    M   7718.7;
      NOT   ;
      =     M   1045.0;
NETWORK
TITLE =
